C05455=1067.841,-44.416,-61.846,172.334,24.240,154.436
C05456=1067.835,-44.665,-61.833,172.333,24.238,154.436
C05457=1067.828,-44.914,-61.820,172.331,24.236,154.436
C05458=1067.822,-45.164,-61.808,172.330,24.234,154.436
C05459=1067.816,-45.414,-61.795,172.328,24.232,154.436
C05460=1067.810,-45.664,-61.783,172.327,24.229,154.435
C05461=1067.804,-45.913,-61.771,172.325,24.227,154.435
C05462=1067.798,-46.163,-61.759,172.324,24.225,154.435
C05463=1067.792,-46.413,-61.746,172.322,24.223,154.435
C05464=1067.786,-46.662,-61.734,172.321,24.221,154.435
C05465=1067.780,-46.912,-61.722,172.320,24.219,154.434
C05466=1067.774,-47.161,-61.709,172.318,24.217,154.434
C05467=1067.768,-47.411,-61.697,172.317,24.215,154.434
C05468=1067.762,-47.661,-61.685,172.315,24.213,154.434
C05469=1067.756,-47.911,-61.672,172.313,24.211,154.434
C05470=1067.749,-48.160,-61.660,172.311,24.208,154.433
C05471=1067.744,-48.409,-61.648,172.310,24.207,154.433
C05472=1067.738,-48.659,-61.636,172.308,24.205,154.433
C05473=1067.732,-48.909,-61.623,172.307,24.202,154.433
C05474=1067.726,-49.159,-61.611,172.305,24.200,154.433
C05475=1067.720,-49.408,-61.599,172.304,24.198,154.432
C05476=1067.713,-49.686,-61.585,172.303,24.196,154.432
C05477=1067.707,-49.963,-61.572,172.301,24.194,154.432
C05478=1067.700,-50.241,-61.558,172.299,24.192,154.432
C05479=1067.693,-50.518,-61.544,172.297,24.189,154.432
C05480=1067.687,-50.767,-61.532,172.296,24.187,154.431
C05481=1067.681,-51.017,-61.520,172.294,24.186,154.431
C05482=1067.674,-51.267,-61.508,172.293,24.184,154.431
C05483=1067.668,-51.516,-61.497,172.292,24.181,154.431
C05484=1067.662,-51.766,-61.484,172.290,24.179,154.431
C05485=1067.656,-52.016,-61.472,172.289,24.178,154.431
C05486=1067.650,-52.266,-61.460,172.287,24.176,154.430
C05487=1067.643,-52.515,-61.448,172.285,24.174,154.430
C05488=1067.637,-52.764,-61.436,172.283,24.172,154.430
C05489=1067.631,-53.014,-61.424,172.282,24.169,154.430
C05490=1067.625,-53.263,-61.412,172.280,24.168,154.430
C05491=1067.618,-53.514,-61.401,172.279,24.166,154.430
C05492=1067.612,-53.764,-61.388,172.277,24.164,154.430
C05493=1067.606,-54.012,-61.376,172.276,24.162,154.429
C05494=1067.600,-54.262,-61.364,172.274,24.160,154.429
C05495=1067.594,-54.512,-61.352,172.273,24.158,154.429
C05496=1067.587,-54.762,-61.341,172.271,24.157,154.429
C05497=1067.582,-55.011,-61.328,172.270,24.154,154.429
C05498=1067.576,-55.261,-61.316,172.268,24.152,154.429
C05499=1067.569,-55.510,-61.305,172.267,24.150,154.428
C05500=1067.563,-55.760,-61.292,172.265,24.149,154.428
C05501=1067.557,-56.010,-61.281,172.264,24.147,154.428
C05502=1067.551,-56.259,-61.269,172.262,24.145,154.428
C05503=1067.545,-56.509,-61.257,172.261,24.143,154.428
C05504=1067.538,-56.759,-61.245,172.259,24.141,154.428
C05505=1067.532,-57.008,-61.234,172.258,24.139,154.427
C05506=1067.526,-57.258,-61.221,172.255,24.137,154.427
C05507=1067.520,-57.508,-61.209,172.254,24.135,154.427
C05508=1067.514,-57.757,-61.198,172.252,24.133,154.427
C05509=1067.508,-58.007,-61.186,172.251,24.131,154.427
C05510=1067.501,-58.257,-61.174,172.249,24.129,154.427
C05511=1067.495,-58.505,-61.162,172.248,24.127,154.427
C05512=1067.490,-58.756,-61.150,172.246,24.126,154.426
C05513=1067.483,-59.006,-61.138,172.245,24.124,154.426
C05514=1067.477,-59.254,-61.127,172.243,24.122,154.426
C05515=1067.471,-59.505,-61.115,172.242,24.120,154.426
C05516=1067.465,-59.755,-61.103,172.240,24.118,154.426
C05517=1067.459,-60.003,-61.091,172.239,24.116,154.426
C05518=1067.453,-60.254,-61.080,172.237,24.115,154.426
C05519=1067.447,-60.503,-61.068,172.236,24.113,154.425
C05520=1067.441,-60.752,-61.056,172.234,24.111,154.425
C05521=1067.434,-61.003,-61.045,172.233,24.109,154.425
C05522=1067.428,-61.252,-61.032,172.231,24.107,154.425
C05523=1067.423,-61.502,-61.021,172.230,24.105,154.425
C05524=1067.416,-61.751,-61.009,172.227,24.103,154.425
C05525=1067.410,-62.001,-60.997,172.226,24.101,154.425
C05526=1067.404,-62.251,-60.986,172.224,24.099,154.424
C05527=1067.398,-62.500,-60.974,172.223,24.098,154.424
C05528=1067.392,-62.750,-60.963,172.221,24.096,154.424
C05529=1067.386,-63.000,-60.951,172.220,24.094,154.424
C05530=1067.380,-63.250,-60.939,172.218,24.092,154.424
C05531=1067.374,-63.499,-60.928,172.217,24.090,154.424
C05532=1067.368,-63.749,-60.916,172.215,24.088,154.424
C05533=1067.362,-63.998,-60.904,172.214,24.087,154.423
C05534=1067.356,-64.248,-60.893,172.212,24.085,154.423
C05535=1067.350,-64.497,-60.881,172.211,24.083,154.423
C05536=1067.344,-64.748,-60.870,172.209,24.081,154.423
C05537=1067.337,-64.997,-60.858,172.208,24.079,154.423
C05538=1067.332,-65.247,-60.847,172.206,24.077,154.423
C05539=1067.325,-65.496,-60.835,172.205,24.076,154.423
C05540=1067.319,-65.775,-60.822,172.202,24.073,154.422
C05541=1067.312,-66.054,-60.809,172.201,24.071,154.422
C05542=1067.305,-66.332,-60.797,172.199,24.069,154.422
C05543=1067.299,-66.611,-60.784,172.198,24.067,154.422
C05544=1067.292,-66.861,-60.772,172.196,24.065,154.422
C05545=1067.287,-67.111,-60.760,172.194,24.063,154.422
C05546=1067.280,-67.360,-60.748,172.192,24.062,154.422
C05547=1067.275,-67.610,-60.738,172.191,24.060,154.422
C05548=1067.268,-67.859,-60.726,172.189,24.058,154.421
C05549=1067.262,-68.109,-60.715,172.188,24.056,154.421
C05550=1067.257,-68.359,-60.703,172.186,24.055,154.421
C05551=1067.251,-68.608,-60.691,172.185,24.053,154.421
C05552=1067.244,-68.858,-60.680,172.183,24.051,154.421
C05553=1067.238,-69.107,-60.668,172.182,24.049,154.421
C05554=1067.232,-69.357,-60.657,172.180,24.047,154.421
C05555=1067.227,-69.607,-60.646,172.179,24.045,154.420
C05556=1067.220,-69.857,-60.634,172.177,24.044,154.420
C05557=1067.214,-70.106,-60.623,172.175,24.042,154.420
C05558=1067.208,-70.357,-60.612,172.174,24.040,154.420
C05559=1067.202,-70.605,-60.600,172.172,24.038,154.420
C05560=1067.196,-70.856,-60.588,172.171,24.037,154.420
C05561=1067.191,-71.105,-60.577,172.169,24.035,154.420
C05562=1067.184,-71.355,-60.565,172.168,24.033,154.419
C05563=1067.178,-71.604,-60.554,172.166,24.032,154.419
C05564=1067.173,-71.854,-60.544,172.165,24.030,154.419
C05565=1067.167,-72.104,-60.531,172.163,24.028,154.419
C05566=1067.161,-72.353,-60.520,172.161,24.026,154.419
C05567=1067.155,-72.604,-60.509,172.159,24.024,154.419
C05568=1067.149,-72.853,-60.498,172.158,24.022,154.419
C05569=1067.142,-73.103,-60.486,172.156,24.021,154.419
C05570=1067.136,-73.352,-60.475,172.155,24.019,154.419
C05571=1067.131,-73.602,-60.464,172.153,24.017,154.419
C05572=1067.125,-73.852,-60.453,172.152,24.015,154.418
C05573=1067.119,-74.101,-60.441,172.150,24.013,154.418
C05574=1067.113,-74.351,-60.430,172.148,24.012,154.418
C05575=1067.107,-74.601,-60.419,172.147,24.010,154.418
C05576=1067.101,-74.851,-60.408,172.145,24.008,154.418
C05577=1067.095,-75.100,-60.397,172.144,24.007,154.418
C05578=1067.088,-75.350,-60.385,172.142,24.005,154.418
C05579=1067.082,-75.599,-60.374,172.141,24.003,154.418
C05580=1067.076,-75.849,-60.364,172.139,24.002,154.418
C05581=1067.070,-76.099,-60.352,172.138,24.000,154.417
C05582=1067.064,-76.348,-60.341,172.136,23.999,154.417
C05583=1067.058,-76.598,-60.330,172.134,23.997,154.417
C05584=1067.052,-76.847,-60.319,172.133,23.995,154.417
C05585=1067.045,-77.097,-60.307,172.131,23.994,154.417
C05586=1067.040,-77.347,-60.296,172.130,23.992,154.417
C05587=1067.034,-77.596,-60.286,172.128,23.990,154.417
C05588=1067.027,-77.847,-60.274,172.126,23.989,154.417
C05589=1067.022,-78.096,-60.263,172.124,23.987,154.417
C05590=1067.015,-78.346,-60.252,172.122,23.986,154.417
C05591=1067.010,-78.596,-60.241,172.121,23.984,154.417
C05592=1067.003,-78.845,-60.231,172.119,23.982,154.416
C05593=1066.997,-79.095,-60.220,172.118,23.981,154.416
C05594=1066.991,-79.344,-60.208,172.116,23.979,154.416
C05595=1066.985,-79.594,-60.197,172.115,23.978,154.416
C05596=1066.979,-79.844,-60.186,172.113,23.976,154.416
C05597=1066.973,-80.093,-60.175,172.111,23.974,154.416
C05598=1066.967,-80.343,-60.164,172.110,23.973,154.416
C05599=1066.960,-80.593,-60.154,172.108,23.971,154.416
C05600=1066.954,-80.843,-60.142,172.107,23.969,154.416
C05601=1066.948,-81.092,-60.132,172.105,23.968,154.416
C05602=1066.942,-81.341,-60.121,172.104,23.966,154.416
C05603=1066.935,-81.592,-60.110,172.102,23.965,154.416
C05604=1066.929,-81.873,-60.098,172.100,23.963,154.415
C05605=1066.922,-82.154,-60.086,172.098,23.962,154.416
C05606=1066.915,-82.435,-60.073,172.096,23.960,154.415
C05607=1066.908,-82.715,-60.062,172.095,23.958,154.415
C05608=1066.902,-82.965,-60.051,172.093,23.957,154.415
C05609=1066.895,-83.215,-60.040,172.092,23.955,154.415
C05610=1066.889,-83.464,-60.029,172.090,23.953,154.415
C05611=1066.883,-83.714,-60.018,172.088,23.952,154.415
C05612=1066.877,-83.964,-60.007,172.086,23.951,154.415
C05613=1066.870,-84.213,-59.997,172.084,23.949,154.415
C05614=1066.864,-84.463,-59.986,172.083,23.947,154.415
C05615=1066.858,-84.713,-59.975,172.081,23.946,154.415
C05616=1066.853,-84.963,-59.965,172.079,23.944,154.415
C05617=1066.846,-85.213,-59.954,172.078,23.943,154.415
C05618=1066.840,-85.462,-59.943,172.076,23.942,154.415
C05619=1066.834,-85.712,-59.932,172.075,23.940,154.415
C05620=1066.827,-85.961,-59.922,172.073,23.939,154.415
C05621=1066.822,-86.211,-59.911,172.071,23.937,154.414
C05622=1066.816,-86.460,-59.900,172.070,23.935,154.414
C05623=1066.809,-86.710,-59.889,172.068,23.934,154.414
C05624=1066.803,-86.960,-59.879,172.066,23.933,154.414
C05625=1066.797,-87.210,-59.869,172.065,23.931,154.414
C05626=1066.791,-87.459,-59.858,172.063,23.930,154.414
C05627=1066.785,-87.709,-59.847,172.062,23.928,154.414
C05628=1066.778,-87.958,-59.836,172.060,23.927,154.414
C05629=1066.773,-88.208,-59.826,172.058,23.925,154.414
C05630=1066.766,-88.459,-59.815,172.057,23.924,154.414
C05631=1066.760,-88.708,-59.805,172.055,23.922,154.414
C05632=1066.754,-88.957,-59.794,172.054,23.921,154.414
C05633=1066.749,-89.207,-59.783,172.052,23.920,154.414
C05634=1066.742,-89.457,-59.773,172.050,23.918,154.414
C05635=1066.736,-89.707,-59.762,172.049,23.916,154.414
C05636=1066.730,-89.956,-59.752,172.047,23.915,154.414
C05637=1066.724,-90.206,-59.741,172.046,23.914,154.414
C05638=1066.718,-90.456,-59.730,172.044,23.913,154.414
C05639=1066.711,-90.706,-59.720,172.042,23.911,154.414
C05640=1066.706,-90.955,-59.709,172.041,23.909,154.413
C05641=1066.700,-91.205,-59.698,172.039,23.908,154.413
C05642=1066.693,-91.455,-59.689,172.037,23.907,154.413
C05643=1066.687,-91.705,-59.678,172.036,23.905,154.413
C05644=1066.681,-91.954,-59.667,172.033,23.903,154.413
C05645=1066.675,-92.204,-59.657,172.032,23.902,154.413
C05646=1066.670,-92.453,-59.646,172.030,23.901,154.413
C05647=1066.663,-92.703,-59.636,172.028,23.900,154.413
C05648=1066.657,-92.953,-59.626,172.027,23.898,154.413
C05649=1066.651,-93.203,-59.615,172.025,23.896,154.413
C05650=1066.645,-93.452,-59.604,172.023,23.895,154.413
C05651=1066.639,-93.702,-59.595,172.022,23.894,154.413
C05652=1066.633,-93.951,-59.584,172.020,23.893,154.413
C05653=1066.627,-94.201,-59.573,172.018,23.891,154.413
C05654=1066.620,-94.451,-59.563,172.017,23.889,154.413
C05655=1066.615,-94.701,-59.552,172.015,23.888,154.413
C05656=1066.608,-94.950,-59.542,172.014,23.887,154.413
C05657=1066.603,-95.200,-59.532,172.012,23.886,154.413
C05658=1066.596,-95.449,-59.521,172.010,23.884,154.413
C05659=1066.590,-95.700,-59.511,172.009,23.883,154.413
C05660=1066.585,-95.950,-59.500,172.007,23.881,154.413
C05661=1066.578,-96.199,-59.490,172.006,23.880,154.413
C05662=1066.573,-96.449,-59.480,172.004,23.879,154.413
C05663=1066.566,-96.698,-59.469,172.002,23.877,154.413
C05664=1066.561,-96.948,-59.459,172.001,23.876,154.413
C05665=1066.554,-97.197,-59.449,171.999,23.875,154.413
C05666=1066.549,-97.447,-59.439,171.997,23.873,154.413
C05667=1066.542,-97.697,-59.428,171.996,23.872,154.413
C05668=1066.535,-97.980,-59.416,171.994,23.871,154.413
C05669=1066.528,-98.264,-59.405,171.991,23.869,154.413
C05670=1066.521,-98.547,-59.393,171.990,23.868,154.413
C05671=1066.514,-98.830,-59.381,171.988,23.866,154.412
C05672=1066.508,-99.080,-59.372,171.986,23.865,154.413
C05673=1066.501,-99.329,-59.362,171.985,23.864,154.413
C05674=1066.496,-99.579,-59.351,171.983,23.863,154.413
C05675=1066.490,-99.828,-59.341,171.981,23.862,154.413
C05676=1066.484,-100.079,-59.331,171.980,23.860,154.413
C05677=1066.477,-100.329,-59.321,171.978,23.859,154.413
C05678=1066.471,-100.578,-59.311,171.976,23.858,154.413
C05679=1066.465,-100.828,-59.301,171.975,23.856,154.412
C05680=1066.459,-101.078,-59.290,171.973,23.855,154.412
C05681=1066.453,-101.327,-59.281,171.971,23.854,154.412
C05682=1066.446,-101.576,-59.271,171.970,23.853,154.412
C05683=1066.441,-101.827,-59.260,171.968,23.851,154.412
C05684=1066.435,-102.076,-59.251,171.966,23.851,154.413
C05685=1066.428,-102.326,-59.240,171.965,23.849,154.413
C05686=1066.422,-102.576,-59.230,171.963,23.848,154.413
C05687=1066.416,-102.826,-59.220,171.961,23.847,154.412
C05688=1066.410,-103.075,-59.210,171.960,23.845,154.412
C05689=1066.404,-103.325,-59.200,171.958,23.844,154.412
C05690=1066.398,-103.575,-59.190,171.956,23.843,154.412
C05691=1066.391,-103.824,-59.180,171.954,23.842,154.413
C05692=1066.386,-104.075,-59.170,171.953,23.841,154.413
C05693=1066.380,-104.324,-59.160,171.951,23.840,154.413
C05694=1066.373,-104.574,-59.150,171.949,23.838,154.413
C05695=1066.367,-104.823,-59.141,171.948,23.837,154.413
C05696=1066.361,-105.073,-59.130,171.946,23.836,154.412
C05697=1066.355,-105.323,-59.120,171.944,23.835,154.413
C05698=1066.349,-105.572,-59.111,171.943,23.834,154.413
C05699=1066.343,-105.822,-59.100,171.941,23.832,154.413
C05700=1066.337,-106.072,-59.090,171.939,23.831,154.413
C05701=1066.331,-106.321,-59.081,171.938,23.830,154.413
C05702=1066.325,-106.571,-59.071,171.936,23.829,154.413
C05703=1066.318,-106.820,-59.061,171.934,23.828,154.413
C05704=1066.312,-107.071,-59.050,171.933,23.827,154.413
C05705=1066.306,-107.321,-59.041,171.931,23.826,154.413
C05706=1066.300,-107.571,-59.031,171.929,23.825,154.413
C05707=1066.294,-107.820,-59.021,171.927,23.823,154.413
C05708=1066.287,-108.070,-59.011,171.926,23.823,154.413
C05709=1066.281,-108.320,-59.002,171.924,23.821,154.413
C05710=1066.275,-108.569,-58.992,171.922,23.820,154.413
C05711=1066.269,-108.819,-58.981,171.920,23.819,154.413
C05712=1066.263,-109.069,-58.972,171.919,23.818,154.413
C05713=1066.257,-109.319,-58.962,171.917,23.817,154.413
C05714=1066.251,-109.568,-58.952,171.915,23.816,154.413
C05715=1066.245,-109.818,-58.943,171.914,23.815,154.413
C05716=1066.238,-110.068,-58.933,171.912,23.813,154.413
C05717=1066.232,-110.317,-58.923,171.910,23.813,154.413
C05718=1066.226,-110.567,-58.913,171.909,23.811,154.413
C05719=1066.220,-110.817,-58.904,171.907,23.811,154.413
C05720=1066.214,-111.067,-58.894,171.905,23.809,154.413
C05721=1066.208,-111.317,-58.884,171.903,23.808,154.413
C05722=1066.202,-111.566,-58.875,171.902,23.807,154.413
C05723=1066.196,-111.816,-58.865,171.900,23.806,154.413
C05724=1066.189,-112.065,-58.855,171.898,23.805,154.413
C05725=1066.183,-112.315,-58.845,171.896,23.804,154.413
C05726=1066.177,-112.565,-58.836,171.895,23.803,154.413
C05727=1066.171,-112.815,-58.826,171.893,23.802,154.413
C05728=1066.165,-113.065,-58.816,171.891,23.801,154.413
C05729=1066.158,-113.314,-58.807,171.889,23.800,154.414
C05730=1066.153,-113.563,-58.798,171.888,23.799,154.414
C05731=1066.147,-113.813,-58.788,171.886,23.798,154.414
C05732=1066.140,-114.095,-58.776,171.883,23.797,154.414
C05733=1066.133,-114.376,-58.766,171.882,23.796,154.414
C05734=1066.126,-114.657,-58.755,171.880,23.795,154.414
C05735=1066.119,-114.939,-58.744,171.878,23.794,154.414
C05736=1066.113,-115.188,-58.735,171.876,23.793,154.414
C05737=1066.107,-115.438,-58.725,171.875,23.792,154.414
C05738=1066.101,-115.687,-58.716,171.873,23.791,154.414
C05739=1066.095,-115.937,-58.706,171.871,23.790,154.414
C05740=1066.088,-116.187,-58.696,171.870,23.789,154.414
C05741=1066.082,-116.437,-58.687,171.868,23.788,154.414
C05742=1066.076,-116.687,-58.677,171.866,23.787,154.414
C05743=1066.070,-116.936,-58.668,171.864,23.786,154.414
C05744=1066.064,-117.186,-58.658,171.862,23.785,154.414
C05745=1066.058,-117.436,-58.649,171.861,23.784,154.414
C05746=1066.051,-117.686,-58.639,171.859,23.783,154.414
C05747=1066.044,-117.935,-58.630,171.857,23.782,154.415
C05748=1066.039,-118.186,-58.621,171.855,23.781,154.415
C05749=1066.033,-118.435,-58.612,171.854,23.780,154.415
C05750=1066.027,-118.685,-58.602,171.852,23.780,154.415
C05751=1066.021,-118.934,-58.593,171.850,23.778,154.415
C05752=1066.015,-119.184,-58.583,171.848,23.778,154.415
C05753=1066.008,-119.434,-58.574,171.847,23.777,154.415
C05754=1066.002,-119.684,-58.564,171.845,23.776,154.415
C05755=1065.996,-119.934,-58.555,171.843,23.775,154.415
C05756=1065.990,-120.183,-58.545,171.841,23.774,154.415
C05757=1065.984,-120.432,-58.536,171.840,23.773,154.415
C05758=1065.978,-120.683,-58.528,171.838,23.772,154.415
C05759=1065.971,-120.932,-58.518,171.836,23.772,154.415
C05760=1065.965,-121.182,-58.508,171.834,23.770,154.415
C05761=1065.959,-121.432,-58.499,171.832,23.770,154.416
C05762=1065.953,-121.682,-58.489,171.831,23.769,154.416
C05763=1065.947,-121.932,-58.480,171.829,23.768,154.416
C05764=1065.941,-122.181,-58.471,171.827,23.767,154.416
C05765=1065.935,-122.431,-58.462,171.825,23.766,154.416
C05766=1065.928,-122.681,-58.453,171.823,23.765,154.416
C05767=1065.922,-122.930,-58.443,171.822,23.765,154.416
C05768=1065.916,-123.180,-58.434,171.820,23.764,154.416
C05769=1065.910,-123.430,-58.424,171.818,23.763,154.416
C05770=1065.905,-123.680,-58.416,171.816,23.762,154.416
C05771=1065.898,-123.929,-58.407,171.815,23.762,154.416
C05772=1065.892,-124.179,-58.397,171.814,23.761,154.416
C05773=1065.885,-124.429,-58.387,171.812,23.760,154.416
C05774=1065.880,-124.679,-58.379,171.810,23.759,154.417
C05775=1065.873,-124.929,-58.369,171.808,23.758,154.417
C05776=1065.867,-125.178,-58.360,171.807,23.757,154.417
C05777=1065.861,-125.428,-58.351,171.805,23.757,154.417
C05778=1065.855,-125.678,-58.342,171.803,23.756,154.417
C05779=1065.849,-125.928,-58.332,171.801,23.755,154.417
C05780=1065.842,-126.177,-58.323,171.799,23.755,154.417
C05781=1065.837,-126.427,-58.315,171.797,23.754,154.417
C05782=1065.831,-126.677,-58.305,171.796,23.753,154.417
C05783=1065.824,-126.926,-58.296,171.794,23.752,154.417
C05784=1065.817,-127.176,-58.287,171.792,23.751,154.418
C05785=1065.812,-127.427,-58.278,171.790,23.750,154.418
C05786=1065.805,-127.675,-58.269,171.788,23.750,154.418
C05787=1065.799,-127.925,-58.260,171.787,23.749,154.418
C05788=1065.795,-128.176,-58.250,171.785,23.748,154.418
C05789=1065.792,-128.427,-58.239,171.784,23.746,154.418
C05790=1065.791,-128.678,-58.228,171.782,23.743,154.417
C05791=1065.791,-128.928,-58.215,171.781,23.740,154.417
C05792=1065.794,-129.181,-58.202,171.781,23.736,154.416
C05793=1065.798,-129.433,-58.189,171.781,23.731,154.416
C05794=1065.804,-129.683,-58.175,171.780,23.726,154.415
C05795=1065.811,-129.934,-58.159,171.780,23.720,154.414
C05796=1065.426,-129.956,-58.337,171.733,23.868,154.446
C05797=1065.418,-129.706,-58.353,171.733,23.875,154.447
C05798=1065.412,-129.455,-58.368,171.733,23.880,154.448
C05799=1065.409,-129.203,-58.381,171.733,23.884,154.449
C05800=1065.406,-128.951,-58.395,171.734,23.888,154.450
C05801=1065.406,-128.700,-58.406,171.735,23.892,154.450
C05802=1065.406,-128.450,-58.418,171.737,23.895,154.451
C05803=1065.410,-128.199,-58.429,171.738,23.896,154.451
C05804=1065.414,-127.948,-58.439,171.740,23.898,154.451
C05805=1065.419,-127.698,-58.448,171.742,23.898,154.451
C05806=1065.426,-127.448,-58.457,171.743,23.900,154.451
C05807=1065.432,-127.198,-58.467,171.745,23.900,154.450
C05808=1065.438,-126.950,-58.475,171.747,23.901,154.450
C05809=1065.444,-126.699,-58.484,171.749,23.902,154.450
C05810=1065.450,-126.449,-58.494,171.751,23.903,154.450
C05811=1065.457,-126.200,-58.503,171.751,23.903,154.450
C05812=1065.462,-125.950,-58.511,171.753,23.904,154.450
C05813=1065.468,-125.700,-58.521,171.755,23.904,154.450
C05814=1065.475,-125.451,-58.530,171.757,23.905,154.450
C05815=1065.482,-125.201,-58.539,171.759,23.906,154.450
C05816=1065.487,-124.951,-58.548,171.761,23.906,154.449
C05817=1065.494,-124.701,-58.558,171.762,23.908,154.450
C05818=1065.499,-124.452,-58.567,171.764,23.908,154.449
C05819=1065.506,-124.202,-58.576,171.766,23.909,154.449
C05820=1065.512,-123.952,-58.585,171.768,23.910,154.449
C05821=1065.518,-123.702,-58.594,171.769,23.911,154.449
C05822=1065.524,-123.452,-58.604,171.771,23.912,154.449
C05823=1065.530,-123.203,-58.613,171.773,23.913,154.449
C05824=1065.536,-122.953,-58.623,171.775,23.913,154.449
C05825=1065.543,-122.703,-58.631,171.777,23.914,154.449
C05826=1065.549,-122.454,-58.640,171.778,23.915,154.449
C05827=1065.555,-122.204,-58.650,171.780,23.916,154.449
C05828=1065.561,-121.954,-58.660,171.782,23.917,154.449
C05829=1065.567,-121.704,-58.669,171.784,23.917,154.448
C05830=1065.573,-121.454,-58.678,171.786,23.918,154.448
C05831=1065.579,-121.205,-58.687,171.787,23.919,154.448
C05832=1065.586,-120.955,-58.696,171.789,23.920,154.448
C05833=1065.592,-120.705,-58.706,171.791,23.921,154.448
C05834=1065.598,-120.456,-58.715,171.793,23.922,154.448
C05835=1065.604,-120.206,-58.725,171.794,23.923,154.448
C05836=1065.610,-119.956,-58.734,171.796,23.923,154.448
C05837=1065.616,-119.707,-58.744,171.798,23.924,154.448
C05838=1065.622,-119.456,-58.753,171.800,23.925,154.448
C05839=1065.628,-119.207,-58.762,171.802,23.926,154.448
C05840=1065.634,-118.957,-58.772,171.803,23.927,154.448
C05841=1065.641,-118.707,-58.781,171.805,23.928,154.448
C05842=1065.647,-118.458,-58.790,171.807,23.929,154.447
C05843=1065.653,-118.208,-58.800,171.808,23.930,154.447
C05844=1065.660,-117.958,-58.809,171.810,23.931,154.447
C05845=1065.666,-117.708,-58.819,171.812,23.931,154.447
C05846=1065.672,-117.458,-58.828,171.814,23.933,154.447
C05847=1065.677,-117.209,-58.838,171.816,23.933,154.447
C05848=1065.684,-116.959,-58.847,171.817,23.934,154.447
C05849=1065.690,-116.710,-58.857,171.819,23.935,154.447
C05850=1065.696,-116.460,-58.866,171.821,23.936,154.447
C05851=1065.702,-116.210,-58.876,171.823,23.937,154.447
C05852=1065.708,-115.960,-58.885,171.824,23.938,154.447
C05853=1065.714,-115.740,-58.893,171.825,23.938,154.447
C05854=1065.719,-115.520,-58.902,171.827,23.940,154.447
C05855=1065.725,-115.300,-58.910,171.829,23.940,154.447
C05856=1065.730,-115.080,-58.919,171.830,23.942,154.447
C05857=1065.736,-114.860,-58.927,171.831,23.942,154.447
C05858=1065.741,-114.639,-58.936,171.833,23.943,154.447
C05859=1065.747,-114.420,-58.944,171.835,23.944,154.447
C05860=1065.751,-114.199,-58.952,171.837,23.945,154.446
C05861=1065.761,-113.836,-58.966,171.839,23.946,154.446
C05862=1065.767,-113.586,-58.976,171.841,23.948,154.446
C05863=1065.773,-113.336,-58.985,171.843,23.948,154.446
C05864=1065.779,-113.086,-58.996,171.844,23.950,154.446
C05865=1065.785,-112.836,-59.005,171.846,23.950,154.446
C05866=1065.791,-112.587,-59.015,171.848,23.952,154.446
C05867=1065.797,-112.337,-59.024,171.850,23.952,154.446
C05868=1065.804,-112.088,-59.035,171.851,23.954,154.446
C05869=1065.810,-111.838,-59.044,171.853,23.955,154.446
C05870=1065.816,-111.588,-59.054,171.855,23.956,154.446
C05871=1065.822,-111.338,-59.063,171.857,23.957,154.446
C05872=1065.828,-111.089,-59.073,171.858,23.958,154.446
C05873=1065.834,-110.839,-59.082,171.860,23.959,154.446
C05874=1065.841,-110.589,-59.092,171.862,23.960,154.446
C05875=1065.846,-110.339,-59.103,171.864,23.961,154.446
C05876=1065.852,-110.090,-59.112,171.865,23.962,154.446
C05877=1065.859,-109.840,-59.122,171.867,23.963,154.446
C05878=1065.865,-109.590,-59.132,171.869,23.964,154.446
C05879=1065.871,-109.340,-59.141,171.870,23.965,154.446
C05880=1065.877,-109.090,-59.151,171.872,23.966,154.446
C05881=1065.884,-108.841,-59.161,171.874,23.967,154.446
C05882=1065.890,-108.591,-59.171,171.876,23.969,154.446
C05883=1065.896,-108.342,-59.180,171.877,23.969,154.446
C05884=1065.901,-108.092,-59.190,171.879,23.971,154.446
C05885=1065.908,-107.842,-59.201,171.881,23.972,154.446
C05886=1065.914,-107.593,-59.210,171.883,23.973,154.446
C05887=1065.920,-107.343,-59.220,171.884,23.974,154.446
C05888=1065.926,-107.093,-59.229,171.886,23.975,154.446
C05889=1065.933,-106.843,-59.239,171.888,23.976,154.445
C05890=1065.938,-106.594,-59.250,171.889,23.977,154.445
C05891=1065.944,-106.344,-59.259,171.891,23.978,154.445
C05892=1065.951,-106.094,-59.269,171.893,23.980,154.445
C05893=1065.957,-105.845,-59.279,171.894,23.980,154.445
C05894=1065.963,-105.595,-59.289,171.896,23.982,154.445
C05895=1065.969,-105.345,-59.299,171.898,23.983,154.445
C05896=1065.976,-105.095,-59.309,171.899,23.984,154.445
C05897=1065.982,-104.845,-59.319,171.901,23.986,154.445
C05898=1065.987,-104.595,-59.329,171.903,23.986,154.445
C05899=1065.994,-104.345,-59.339,171.905,23.988,154.445
C05900=1066.000,-104.096,-59.349,171.906,23.989,154.445
C05901=1066.006,-103.846,-59.359,171.908,23.990,154.445
C05902=1066.012,-103.597,-59.370,171.910,23.991,154.445
C05903=1066.018,-103.347,-59.379,171.911,23.993,154.445
C05904=1066.024,-103.097,-59.389,171.913,23.993,154.445
C05905=1066.030,-102.848,-59.400,171.915,23.995,154.445
C05906=1066.036,-102.598,-59.409,171.916,23.996,154.445
C05907=1066.042,-102.348,-59.419,171.918,23.997,154.445
C05908=1066.048,-102.099,-59.430,171.920,23.998,154.445
C05909=1066.055,-101.848,-59.439,171.921,24.000,154.445
C05910=1066.061,-101.599,-59.450,171.923,24.001,154.445
C05911=1066.067,-101.349,-59.460,171.925,24.002,154.445
C05912=1066.073,-101.099,-59.469,171.927,24.003,154.445
C05913=1066.079,-100.850,-59.480,171.928,24.004,154.445
C05914=1066.085,-100.600,-59.490,171.930,24.006,154.445
C05915=1066.091,-100.351,-59.500,171.932,24.007,154.445
C05916=1066.098,-100.101,-59.510,171.933,24.008,154.445
C05917=1066.103,-99.851,-59.521,171.935,24.009,154.445
C05918=1066.110,-99.601,-59.531,171.937,24.011,154.445
C05919=1066.117,-99.352,-59.541,171.938,24.012,154.445
C05920=1066.122,-99.102,-59.551,171.940,24.013,154.445
C05921=1066.128,-98.853,-59.561,171.942,24.015,154.445
C05922=1066.135,-98.569,-59.572,171.943,24.016,154.445
C05923=1066.143,-98.286,-59.584,171.946,24.017,154.445
C05924=1066.149,-98.003,-59.596,171.948,24.019,154.445
C05925=1066.156,-97.719,-59.607,171.949,24.020,154.445
C05926=1066.163,-97.469,-59.618,171.951,24.021,154.445
C05927=1066.168,-97.219,-59.628,171.953,24.023,154.445
C05928=1066.175,-96.970,-59.638,171.954,24.024,154.445
C05929=1066.180,-96.720,-59.648,171.956,24.026,154.446
C05930=1066.187,-96.471,-59.659,171.957,24.027,154.446
C05931=1066.192,-96.221,-59.670,171.959,24.028,154.446
C05932=1066.199,-95.971,-59.679,171.961,24.029,154.446
C05933=1066.204,-95.722,-59.690,171.962,24.031,154.446
C05934=1066.210,-95.471,-59.701,171.964,24.032,154.446
C05935=1066.217,-95.222,-59.711,171.966,24.033,154.446
C05936=1066.223,-94.972,-59.722,171.967,24.035,154.446
C05937=1066.229,-94.722,-59.731,171.969,24.036,154.446
C05938=1066.235,-94.473,-59.742,171.971,24.038,154.446
C05939=1066.241,-94.223,-59.752,171.972,24.039,154.446
C05940=1066.247,-93.973,-59.763,171.974,24.040,154.446
C05941=1066.253,-93.724,-59.774,171.976,24.042,154.446
C05942=1066.259,-93.474,-59.783,171.978,24.043,154.446
C05943=1066.265,-93.224,-59.794,171.980,24.045,154.446
C05944=1066.271,-92.975,-59.805,171.981,24.046,154.446
C05945=1066.277,-92.724,-59.815,171.983,24.048,154.446
C05946=1066.284,-92.475,-59.825,171.985,24.049,154.446
C05947=1066.289,-92.226,-59.836,171.986,24.050,154.446
C05948=1066.295,-91.975,-59.846,171.988,24.052,154.446
C05949=1066.301,-91.726,-59.857,171.989,24.053,154.446
C05950=1066.308,-91.476,-59.868,171.991,24.054,154.446
C05951=1066.314,-91.226,-59.878,171.993,24.056,154.446
C05952=1066.320,-90.977,-59.888,171.994,24.058,154.446
C05953=1066.325,-90.727,-59.899,171.996,24.059,154.446
C05954=1066.332,-90.478,-59.910,171.998,24.060,154.446
C05955=1066.338,-90.227,-59.920,171.999,24.061,154.446
C05956=1066.344,-89.978,-59.931,172.001,24.063,154.447
C05957=1066.350,-89.729,-59.941,172.002,24.065,154.447
C05958=1066.356,-89.479,-59.952,172.004,24.066,154.447
C05959=1066.363,-89.229,-59.962,172.006,24.067,154.447
C05960=1066.368,-88.979,-59.973,172.007,24.069,154.447
C05961=1066.374,-88.730,-59.984,172.009,24.070,154.447
C05962=1066.381,-88.480,-59.995,172.011,24.072,154.447
C05963=1066.387,-88.230,-60.005,172.012,24.073,154.447
C05964=1066.392,-87.980,-60.016,172.014,24.075,154.447
C05965=1066.399,-87.731,-60.026,172.016,24.076,154.447
C05966=1066.405,-87.481,-60.037,172.017,24.077,154.447
C05967=1066.411,-87.231,-60.048,172.019,24.079,154.447
C05968=1066.417,-86.982,-60.058,172.020,24.080,154.447
C05969=1066.424,-86.732,-60.069,172.022,24.082,154.447
C05970=1066.430,-86.482,-60.079,172.024,24.083,154.447
C05971=1066.436,-86.233,-60.090,172.025,24.085,154.447
C05972=1066.442,-85.982,-60.101,172.027,24.086,154.447
C05973=1066.448,-85.733,-60.111,172.028,24.088,154.448
C05974=1066.454,-85.484,-60.122,172.031,24.089,154.447
C05975=1066.460,-85.234,-60.134,172.033,24.091,154.448
C05976=1066.467,-84.984,-60.144,172.034,24.093,154.448
C05977=1066.473,-84.735,-60.155,172.036,24.094,154.448
C05978=1066.479,-84.485,-60.166,172.037,24.096,154.448
C05979=1066.484,-84.235,-60.176,172.039,24.097,154.448
C05980=1066.491,-83.985,-60.186,172.041,24.098,154.448
C05981=1066.497,-83.735,-60.198,172.042,24.100,154.448
C05982=1066.503,-83.486,-60.209,172.044,24.101,154.448
C05983=1066.510,-83.237,-60.219,172.046,24.103,154.448
C05984=1066.516,-82.986,-60.230,172.047,24.104,154.448
C05985=1066.522,-82.737,-60.241,172.049,24.106,154.448
C05986=1066.530,-82.456,-60.253,172.050,24.108,154.448
C05987=1066.536,-82.175,-60.265,172.053,24.109,154.448
C05988=1066.543,-81.894,-60.278,172.054,24.111,154.448
C05989=1066.550,-81.613,-60.290,172.056,24.113,154.449
C05990=1066.556,-81.363,-60.300,172.057,24.114,154.449
C05991=1066.563,-81.113,-60.311,172.059,24.115,154.449
C05992=1066.568,-80.864,-60.322,172.061,24.117,154.449
C05993=1066.574,-80.614,-60.333,172.062,24.119,154.449
C05994=1066.581,-80.364,-60.344,172.064,24.120,154.449
C05995=1066.587,-80.115,-60.354,172.066,24.122,154.449
C05996=1066.593,-79.865,-60.366,172.067,24.123,154.449
C05997=1066.599,-79.616,-60.377,172.069,24.125,154.449
C05998=1066.605,-79.366,-60.388,172.071,24.127,154.449
C05999=1066.611,-79.116,-60.399,172.073,24.128,154.449
C06000=1066.617,-78.867,-60.410,172.074,24.130,154.449
C06001=1066.624,-78.616,-60.421,172.076,24.132,154.449
C06002=1066.630,-78.367,-60.432,172.078,24.133,154.449
C06003=1066.636,-78.118,-60.443,172.079,24.135,154.450
C06004=1066.642,-77.868,-60.454,172.081,24.136,154.450
C06005=1066.648,-77.618,-60.465,172.082,24.138,154.450
C06006=1066.654,-77.368,-60.476,172.084,24.140,154.450
C06007=1066.660,-77.118,-60.487,172.085,24.141,154.450
C06008=1066.666,-76.870,-60.498,172.087,24.143,154.450
C06009=1066.672,-76.619,-60.510,172.088,24.145,154.450
C06010=1066.678,-76.370,-60.521,172.090,24.146,154.450
C06011=1066.684,-76.120,-60.532,172.092,24.148,154.450
C06012=1066.690,-75.870,-60.543,172.093,24.150,154.451
C06013=1066.696,-75.620,-60.554,172.095,24.151,154.451
C06014=1066.703,-75.371,-60.566,172.096,24.153,154.451
C06015=1066.708,-75.122,-60.576,172.098,24.154,154.451
C06016=1066.715,-74.871,-60.588,172.099,24.156,154.451
C06017=1066.720,-74.622,-60.599,172.101,24.158,154.451
C06018=1066.727,-74.372,-60.609,172.103,24.159,154.451
C06019=1066.733,-74.123,-60.621,172.104,24.161,154.451
C06020=1066.740,-73.873,-60.632,172.106,24.163,154.451
C06021=1066.745,-73.623,-60.643,172.108,24.165,154.451
C06022=1066.751,-73.373,-60.655,172.110,24.167,154.452
C06023=1066.757,-73.124,-60.666,172.111,24.168,154.452
C06024=1066.763,-72.875,-60.677,172.113,24.170,154.452
C06025=1066.769,-72.625,-60.688,172.114,24.172,154.452
C06026=1066.775,-72.375,-60.699,172.116,24.174,154.452
C06027=1066.781,-72.125,-60.712,172.117,24.176,154.452
C06028=1066.787,-71.876,-60.723,172.119,24.177,154.452
C06029=1066.793,-71.625,-60.734,172.121,24.179,154.452
C06030=1066.799,-71.377,-60.746,172.122,24.181,154.452
C06031=1066.805,-71.127,-60.756,172.124,24.182,154.453
C06032=1066.810,-70.877,-60.768,172.125,24.184,154.453
C06033=1066.816,-70.628,-60.780,172.127,24.186,154.453
C06034=1066.823,-70.378,-60.791,172.128,24.188,154.453
C06035=1066.828,-70.128,-60.802,172.130,24.190,154.453
C06036=1066.835,-69.878,-60.814,172.131,24.191,154.453
C06037=1066.841,-69.629,-60.825,172.133,24.193,154.453
C06038=1066.846,-69.378,-60.837,172.134,24.195,154.453
C06039=1066.853,-69.130,-60.848,172.136,24.197,154.454
C06040=1066.859,-68.879,-60.860,172.137,24.198,154.454
C06041=1066.865,-68.630,-60.870,172.139,24.200,154.454
C06042=1066.871,-68.380,-60.883,172.141,24.202,154.454
C06043=1066.876,-68.131,-60.894,172.143,24.204,154.454
C06044=1066.883,-67.881,-60.906,172.144,24.206,154.454
C06045=1066.889,-67.631,-60.917,172.146,24.208,154.454
C06046=1066.895,-67.382,-60.929,172.147,24.210,154.455
C06047=1066.900,-67.132,-60.940,172.149,24.211,154.455
C06048=1066.907,-66.882,-60.951,172.151,24.213,154.455
C06049=1066.913,-66.633,-60.963,172.152,24.215,154.455
C06050=1066.920,-66.353,-60.976,172.154,24.216,154.455
C06051=1066.926,-66.075,-60.989,172.155,24.219,154.455
C06052=1066.933,-65.796,-61.002,172.157,24.221,154.455
C06053=1066.940,-65.517,-61.014,172.159,24.223,154.455
C06054=1066.946,-65.268,-61.026,172.160,24.225,154.456
C06055=1066.951,-65.018,-61.038,172.162,24.227,154.456
C06056=1066.958,-64.768,-61.050,172.164,24.228,154.456
C06057=1066.964,-64.518,-61.061,172.165,24.230,154.456
C06058=1066.970,-64.269,-61.073,172.167,24.232,154.456
C06059=1066.976,-64.019,-61.084,172.168,24.234,154.456
C06060=1066.982,-63.770,-61.096,172.170,24.236,154.456
C06061=1066.988,-63.520,-61.107,172.171,24.238,154.457
C06062=1066.994,-63.271,-61.119,172.173,24.239,154.457
C06063=1067.000,-63.020,-61.131,172.175,24.242,154.457
C06064=1067.006,-62.771,-61.143,172.177,24.243,154.457
C06065=1067.013,-62.522,-61.154,172.178,24.245,154.457
C06066=1067.019,-62.272,-61.165,172.180,24.247,154.457
C06067=1067.024,-62.023,-61.178,172.181,24.249,154.457
C06068=1067.031,-61.772,-61.189,172.183,24.251,154.458
C06069=1067.037,-61.523,-61.201,172.184,24.253,154.458
C06070=1067.042,-61.274,-61.213,172.186,24.254,154.458
C06071=1067.049,-61.024,-61.224,172.187,24.256,154.458
C06072=1067.055,-60.774,-61.236,172.189,24.258,154.458
C06073=1067.061,-60.524,-61.247,172.190,24.260,154.458
C06074=1067.067,-60.275,-61.260,172.192,24.262,154.458
C06075=1067.074,-60.025,-61.272,172.193,24.264,154.459
C06076=1067.079,-59.776,-61.283,172.195,24.265,154.459
C06077=1067.085,-59.526,-61.295,172.196,24.267,154.459
C06078=1067.092,-59.276,-61.307,172.198,24.269,154.459
C06079=1067.098,-59.027,-61.318,172.199,24.271,154.459
C06080=1067.104,-58.777,-61.330,172.201,24.273,154.459
C06081=1067.110,-58.527,-61.342,172.202,24.275,154.459
C06082=1067.116,-58.278,-61.353,172.205,24.277,154.460
C06083=1067.122,-58.028,-61.366,172.206,24.279,154.460
C06084=1067.129,-57.778,-61.378,172.208,24.281,154.460
C06085=1067.135,-57.529,-61.389,172.209,24.283,154.460
C06086=1067.140,-57.279,-61.401,172.211,24.285,154.460
C06087=1067.147,-57.029,-61.413,172.212,24.287,154.460
C06088=1067.154,-56.780,-61.425,172.214,24.288,154.461
C06089=1067.159,-56.530,-61.437,172.215,24.290,154.461
C06090=1067.165,-56.280,-61.449,172.217,24.292,154.461
C06091=1067.172,-56.031,-61.461,172.218,24.294,154.461
C06092=1067.178,-55.781,-61.473,172.220,24.296,154.461
C06093=1067.184,-55.532,-61.485,172.221,24.298,154.461
C06094=1067.190,-55.282,-61.496,172.223,24.300,154.462
C06095=1067.196,-55.032,-61.508,172.224,24.302,154.462
C06096=1067.203,-54.782,-61.520,172.226,24.304,154.462
C06097=1067.209,-54.533,-61.532,172.227,24.305,154.462
C06098=1067.215,-54.284,-61.545,172.229,24.307,154.462
C06099=1067.221,-54.033,-61.556,172.230,24.309,154.462
C06100=1067.227,-53.783,-61.568,172.232,24.311,154.462
C06101=1067.233,-53.535,-61.580,172.234,24.314,154.463
C06102=1067.240,-53.285,-61.592,172.236,24.316,154.463
C06103=1067.246,-53.035,-61.605,172.237,24.317,154.463
C06104=1067.252,-52.786,-61.616,172.239,24.319,154.463
C06105=1067.259,-52.535,-61.628,172.240,24.321,154.463
C06106=1067.264,-52.286,-61.640,172.242,24.323,154.463
C06107=1067.270,-52.037,-61.652,172.243,24.325,154.464
C06108=1067.276,-51.787,-61.664,172.245,24.327,154.464
C06109=1067.283,-51.537,-61.676,172.246,24.329,154.464
C06110=1067.290,-51.288,-61.688,172.248,24.331,154.464
C06111=1067.295,-51.038,-61.701,172.249,24.333,154.464
C06112=1067.302,-50.789,-61.712,172.251,24.334,154.464
C06113=1067.308,-50.539,-61.725,172.252,24.337,154.465
C06114=1067.315,-50.261,-61.738,172.254,24.339,154.465
C06115=1067.321,-49.984,-61.752,172.256,24.341,154.465
C06116=1067.328,-49.706,-61.766,172.258,24.343,154.465
C06117=1067.334,-49.429,-61.779,172.259,24.346,154.465
C06118=1067.341,-49.179,-61.791,172.260,24.347,154.466
C06119=1067.347,-48.929,-61.803,172.262,24.350,154.466
C06120=1067.352,-48.680,-61.816,172.264,24.352,154.466
C06121=1067.359,-48.430,-61.828,172.266,24.354,154.466
C06122=1067.365,-48.181,-61.840,172.267,24.356,154.466
C06123=1067.370,-47.931,-61.853,172.269,24.358,154.466
C06124=1067.377,-47.681,-61.865,172.270,24.360,154.467
C06125=1067.382,-47.432,-61.877,172.272,24.362,154.467
C06126=1067.388,-47.182,-61.889,172.273,24.364,154.467
C06127=1067.394,-46.932,-61.902,172.274,24.367,154.467
C06128=1067.401,-46.683,-61.914,172.276,24.368,154.467
C06129=1067.407,-46.433,-61.926,172.277,24.371,154.468
C06130=1067.412,-46.183,-61.939,172.279,24.373,154.468
C06131=1067.419,-45.935,-61.951,172.280,24.375,154.468
C06132=1067.425,-45.685,-61.964,172.282,24.377,154.468
C06133=1067.431,-45.435,-61.976,172.283,24.379,154.468
C06134=1067.437,-45.185,-61.988,172.285,24.381,154.469
C06135=1067.443,-44.935,-62.001,172.286,24.383,154.469
C06136=1067.449,-44.686,-62.013,172.288,24.385,154.469
C06137=1067.455,-44.436,-62.026,172.289,24.387,154.469
C06138=1067.461,-44.187,-62.038,172.290,24.389,154.470
C06139=1067.467,-43.937,-62.050,172.293,24.392,154.470
C06140=1067.473,-43.688,-62.063,172.294,24.393,154.470
C06141=1067.479,-43.438,-62.076,172.296,24.396,154.470
C06142=1067.486,-43.188,-62.088,172.297,24.398,154.470
C06143=1067.491,-42.939,-62.100,172.299,24.400,154.470
C06144=1067.497,-42.689,-62.113,172.300,24.402,154.471
C06145=1067.503,-42.439,-62.125,172.302,24.404,154.471
C06146=1067.510,-42.190,-62.138,172.303,24.406,154.471
C06147=1067.516,-41.940,-62.151,172.305,24.409,154.471
C06148=1067.522,-41.690,-62.163,172.306,24.410,154.471
C06149=1067.528,-41.440,-62.176,172.307,24.413,154.472
C06150=1067.534,-41.191,-62.188,172.309,24.415,154.472
C06151=1067.541,-40.942,-62.201,172.310,24.417,154.472
C06152=1067.546,-40.692,-62.213,172.312,24.419,154.472
C06153=1067.552,-40.443,-62.226,172.313,24.421,154.472
C06154=1067.558,-40.193,-62.238,172.315,24.423,154.473
C06155=1067.565,-39.944,-62.251,172.316,24.425,154.473
C06156=1067.571,-39.694,-62.263,172.318,24.427,154.473
C06157=1067.576,-39.444,-62.276,172.319,24.429,154.473
C06158=1067.582,-39.194,-62.288,172.322,24.432,154.473
C06159=1067.589,-38.945,-62.301,172.323,24.434,154.474
C06160=1067.595,-38.695,-62.314,172.324,24.436,154.474
C06161=1067.601,-38.445,-62.326,172.326,24.438,154.474
C06162=1067.607,-38.196,-62.340,172.327,24.440,154.474
C06163=1067.613,-37.946,-62.352,172.329,24.443,154.475
C06164=1067.619,-37.696,-62.365,172.330,24.444,154.475
C06165=1067.625,-37.447,-62.378,172.332,24.447,154.475
C06166=1067.631,-37.198,-62.390,172.333,24.449,154.475
C06167=1067.637,-36.948,-62.403,172.335,24.451,154.475
C06168=1067.643,-36.699,-62.416,172.336,24.453,154.476
C06169=1067.649,-36.449,-62.428,172.337,24.456,154.476
C06170=1067.655,-36.199,-62.441,172.339,24.458,154.476
C06171=1067.661,-35.950,-62.454,172.340,24.460,154.476
C06172=1067.667,-35.700,-62.467,172.342,24.462,154.476
C06173=1067.673,-35.450,-62.479,172.343,24.464,154.477
C06174=1067.679,-35.201,-62.493,172.344,24.467,154.477
C06175=1067.685,-34.951,-62.505,172.346,24.468,154.477
C06176=1067.691,-34.702,-62.518,172.347,24.471,154.477
C06177=1067.697,-34.452,-62.531,172.349,24.473,154.478
C06178=1067.703,-34.175,-62.545,172.351,24.476,154.478
C06179=1067.710,-33.898,-62.560,172.352,24.478,154.478
C06180=1067.717,-33.621,-62.574,172.354,24.481,154.478
C06181=1067.724,-33.343,-62.588,172.356,24.483,154.479
C06182=1067.730,-33.094,-62.601,172.358,24.485,154.479
C06183=1067.736,-32.844,-62.614,172.359,24.488,154.479
C06184=1067.742,-32.594,-62.627,172.360,24.490,154.479
C06185=1067.748,-32.345,-62.640,172.362,24.492,154.480
C06186=1067.754,-32.095,-62.653,172.363,24.494,154.480
C06187=1067.760,-31.846,-62.666,172.365,24.497,154.480
C06188=1067.766,-31.596,-62.678,172.366,24.498,154.480
C06189=1067.772,-31.347,-62.692,172.368,24.501,154.481
C06190=1067.778,-31.097,-62.704,172.369,24.503,154.481
C06191=1067.785,-30.848,-62.718,172.371,24.505,154.481
C06192=1067.791,-30.598,-62.730,172.372,24.507,154.481
C06193=1067.797,-30.349,-62.743,172.373,24.510,154.481
C06194=1067.803,-30.099,-62.756,172.375,24.512,154.482
C06195=1067.809,-29.849,-62.769,172.376,24.514,154.482
C06196=1067.815,-29.600,-62.782,172.378,24.516,154.482
C06197=1067.821,-29.350,-62.795,172.379,24.519,154.482
C06198=1067.826,-29.101,-62.809,172.381,24.521,154.483
C06199=1067.832,-28.851,-62.821,172.382,24.523,154.483
C06200=1067.839,-28.601,-62.835,172.384,24.526,154.483
C06201=1067.845,-28.351,-62.848,172.386,24.528,154.483
C06202=1067.851,-28.102,-62.861,172.387,24.530,154.483
C06203=1067.858,-27.852,-62.874,172.389,24.532,154.484
C06204=1067.863,-27.603,-62.887,172.390,24.535,154.484
C06205=1067.870,-27.353,-62.900,172.391,24.537,154.484
C06206=1067.876,-27.104,-62.913,172.393,24.539,154.484
C06207=1067.882,-26.854,-62.926,172.394,24.541,154.485
C06208=1067.888,-26.605,-62.939,172.396,24.544,154.485
C06209=1067.893,-26.355,-62.953,172.397,24.546,154.485
C06210=1067.899,-26.105,-62.965,172.399,24.548,154.485
C06211=1067.906,-25.856,-62.979,172.400,24.550,154.486
C06212=1067.912,-25.606,-62.992,172.401,24.553,154.486
C06213=1067.918,-25.356,-63.006,172.403,24.555,154.486
C06214=1067.924,-25.107,-63.019,172.404,24.557,154.487
C06215=1067.930,-24.858,-63.032,172.405,24.560,154.487
C06216=1067.935,-24.607,-63.045,172.407,24.562,154.487
C06217=1067.941,-24.358,-63.058,172.408,24.564,154.487
C06218=1067.948,-24.109,-63.072,172.410,24.566,154.487
C06219=1067.954,-23.860,-63.085,172.411,24.569,154.488
C06220=1067.959,-23.609,-63.098,172.413,24.571,154.488
C06221=1067.965,-23.360,-63.111,172.415,24.574,154.488
C06222=1067.971,-23.111,-63.125,172.416,24.576,154.489
C06223=1067.977,-22.861,-63.139,172.418,24.579,154.489
C06224=1067.984,-22.611,-63.152,172.419,24.581,154.489
C06225=1067.990,-22.361,-63.165,172.420,24.583,154.489
C06226=1067.996,-22.112,-63.178,172.422,24.585,154.489
C06227=1068.001,-21.863,-63.192,172.423,24.588,154.490
C06228=1068.007,-21.613,-63.205,172.425,24.590,154.490
C06229=1068.014,-21.364,-63.218,172.426,24.592,154.490
C06230=1068.019,-21.113,-63.232,172.428,24.595,154.491
C06231=1068.026,-20.864,-63.245,172.429,24.597,154.491
C06232=1068.032,-20.615,-63.258,172.430,24.600,154.491
C06233=1068.037,-20.365,-63.272,172.432,24.602,154.491
C06234=1068.044,-20.116,-63.286,172.433,24.604,154.492
C06235=1068.050,-19.866,-63.299,172.435,24.606,154.492
C06236=1068.056,-19.616,-63.313,172.436,24.608,154.492
C06237=1068.062,-19.366,-63.326,172.437,24.611,154.492
C06238=1068.068,-19.117,-63.339,172.439,24.613,154.493
C06239=1068.073,-18.867,-63.353,172.440,24.616,154.493
C06240=1068.080,-18.618,-63.366,172.442,24.618,154.493
C06241=1068.086,-18.369,-63.379,172.443,24.620,154.493
C06242=1068.093,-18.091,-63.395,172.445,24.623,154.494
C06243=1068.099,-17.813,-63.410,172.447,24.625,154.494
C06244=1068.106,-17.534,-63.425,172.448,24.628,154.494
C06245=1068.113,-17.257,-63.440,172.449,24.631,154.495
C06246=1068.119,-17.007,-63.454,172.452,24.633,154.495
C06247=1068.125,-16.758,-63.467,172.453,24.636,154.495
C06248=1068.132,-16.508,-63.481,172.454,24.638,154.495
C06249=1068.137,-16.259,-63.495,172.456,24.641,154.496
C06250=1068.143,-16.009,-63.508,172.457,24.643,154.496
C06251=1068.150,-15.760,-63.521,172.459,24.645,154.496
C06252=1068.156,-15.510,-63.535,172.460,24.647,154.496
C06253=1068.162,-15.261,-63.549,172.461,24.650,154.497
C06254=1068.167,-15.011,-63.562,172.463,24.652,154.497
C06255=1068.174,-14.762,-63.576,172.464,24.654,154.497
C06256=1068.180,-14.511,-63.590,172.466,24.657,154.497
C06257=1068.186,-14.262,-63.603,172.467,24.659,154.498
C06258=1068.191,-14.013,-63.617,172.468,24.662,154.498
C06259=1068.198,-13.763,-63.630,172.470,24.664,154.498
C06260=1068.204,-13.513,-63.645,172.471,24.667,154.499
C06261=1068.209,-13.263,-63.658,172.472,24.669,154.499
C06262=1068.215,-13.014,-63.672,172.474,24.672,154.499
C06263=1068.221,-12.765,-63.686,172.475,24.674,154.499
C06264=1068.227,-12.515,-63.699,172.477,24.676,154.500
C06265=1068.233,-12.266,-63.714,172.478,24.679,154.500
C06266=1068.240,-12.016,-63.727,172.479,24.681,154.500
C06267=1068.245,-11.767,-63.741,172.481,24.683,154.501
C06268=1068.251,-11.517,-63.755,172.482,24.686,154.501
C06269=1068.257,-11.267,-63.768,172.484,24.688,154.501
C06270=1068.263,-11.018,-63.782,172.485,24.691,154.501
C06271=1068.269,-10.768,-63.796,172.487,24.693,154.502
C06272=1068.275,-10.519,-63.811,172.489,24.696,154.502
C06273=1068.281,-10.269,-63.824,172.490,24.699,154.502
C06274=1068.287,-10.020,-63.838,172.491,24.701,154.503
C06275=1068.293,-9.770,-63.852,172.493,24.703,154.503
C06276=1068.299,-9.520,-63.865,172.494,24.706,154.503
C06277=1068.305,-9.271,-63.879,172.496,24.708,154.503
C06278=1068.311,-9.022,-63.894,172.497,24.710,154.504
C06279=1068.317,-8.772,-63.907,172.498,24.713,154.504
C06280=1068.323,-8.522,-63.921,172.500,24.715,154.504
C06281=1068.328,-8.273,-63.935,172.501,24.718,154.504
C06282=1068.336,-8.023,-63.949,172.503,24.720,154.505
C06283=1068.341,-7.774,-63.963,172.504,24.722,154.505
C06284=1068.347,-7.525,-63.976,172.505,24.725,154.505
C06285=1068.353,-7.274,-63.991,172.507,24.728,154.506
C06286=1068.359,-7.025,-64.005,172.508,24.730,154.506
C06287=1068.365,-6.776,-64.019,172.509,24.732,154.506
C06288=1068.371,-6.526,-64.033,172.511,24.735,154.507
C06289=1068.377,-6.276,-64.047,172.512,24.737,154.507
C06290=1068.383,-6.028,-64.061,172.514,24.739,154.507
C06291=1068.389,-5.777,-64.075,172.515,24.742,154.507
C06292=1068.395,-5.528,-64.089,172.516,24.744,154.508
C06293=1068.402,-5.278,-64.103,172.518,24.747,154.508
C06294=1068.408,-5.029,-64.117,172.519,24.749,154.508
C06295=1068.413,-4.779,-64.131,172.521,24.751,154.508
C06296=1068.420,-4.530,-64.145,172.522,24.754,154.509
C06297=1068.426,-4.280,-64.159,172.523,24.757,154.509
C06298=1068.432,-4.030,-64.173,172.526,24.759,154.509
C06299=1068.438,-3.781,-64.187,172.527,24.762,154.510
C06300=1068.444,-3.532,-64.201,172.528,24.764,154.510
C06301=1068.450,-3.282,-64.216,172.530,24.766,154.510
C06302=1068.456,-3.033,-64.230,172.531,24.769,154.510
C06303=1068.462,-2.783,-64.243,172.532,24.772,154.511
C06304=1068.468,-2.534,-64.258,172.534,24.774,154.511
C06305=1068.474,-2.284,-64.272,172.535,24.776,154.511
C06306=1068.480,-2.004,-64.288,172.537,24.779,154.512
C06307=1068.487,-1.725,-64.304,172.538,24.782,154.512
C06308=1068.493,-1.446,-64.320,172.540,24.785,154.512
C06309=1068.500,-1.166,-64.336,172.541,24.788,154.513
C06310=1068.506,-0.916,-64.351,172.543,24.790,154.513
C06311=1068.511,-0.667,-64.365,172.544,24.793,154.513
C06312=1068.517,-0.418,-64.379,172.545,24.796,154.514
C06313=1068.523,-0.167,-64.394,172.547,24.798,154.514
C06314=1068.530,0.081,-64.408,172.548,24.800,154.514
C06315=1068.536,0.332,-64.422,172.550,24.803,154.515
C06316=1068.542,0.581,-64.436,172.551,24.806,154.515
C06317=1068.547,0.830,-64.450,172.552,24.808,154.515
C06318=1068.554,1.080,-64.465,172.554,24.810,154.515
C06319=1068.559,1.329,-64.479,172.555,24.813,154.516
C06320=1068.565,1.579,-64.494,172.556,24.816,154.516
C06321=1068.571,1.829,-64.508,172.558,24.818,154.516
C06322=1068.577,2.078,-64.522,172.559,24.820,154.517
C06323=1068.583,2.327,-64.537,172.561,24.823,154.517
C06324=1068.589,2.577,-64.551,172.562,24.826,154.517
C06325=1068.595,2.826,-64.566,172.563,24.828,154.518
C06326=1068.600,3.076,-64.580,172.565,24.830,154.518
C06327=1068.607,3.326,-64.595,172.566,24.833,154.518
C06328=1068.612,3.575,-64.609,172.567,24.836,154.519
C06329=1068.619,3.825,-64.624,172.570,24.838,154.519
C06330=1068.624,4.074,-64.638,172.571,24.841,154.519
C06331=1068.630,4.323,-64.652,172.572,24.844,154.520
C06332=1068.636,4.573,-64.667,172.574,24.846,154.520
C06333=1068.642,4.822,-64.682,172.575,24.848,154.520
C06334=1068.648,5.072,-64.696,172.577,24.851,154.520
C06335=1068.654,5.321,-64.711,172.578,24.854,154.521
C06336=1068.660,5.571,-64.726,172.579,24.856,154.521
C06337=1068.666,5.821,-64.739,172.581,24.858,154.521
C06338=1068.672,6.070,-64.754,172.582,24.861,154.522
C06339=1068.678,6.319,-64.769,172.583,24.864,154.522
C06340=1068.684,6.569,-64.783,172.585,24.866,154.522
C06341=1068.690,6.818,-64.798,172.586,24.868,154.523
C06342=1068.696,7.068,-64.813,172.587,24.871,154.523
C06343=1068.702,7.318,-64.827,172.589,24.874,154.523
C06344=1068.708,7.567,-64.842,172.590,24.876,154.523
C06345=1068.714,7.817,-64.856,172.591,24.879,154.524
C06346=1068.720,8.066,-64.871,172.593,24.881,154.524
C06347=1068.726,8.316,-64.885,172.594,24.884,154.524
C06348=1068.732,8.565,-64.900,172.596,24.886,154.525
C06349=1068.738,8.815,-64.915,172.597,24.889,154.525
C06350=1068.744,9.064,-64.929,172.598,24.891,154.525
C06351=1068.750,9.314,-64.944,172.600,24.894,154.526
C06352=1068.756,9.563,-64.958,172.601,24.897,154.526
C06353=1068.762,9.813,-64.973,172.602,24.899,154.526
C06354=1068.769,10.062,-64.988,172.604,24.901,154.527
C06355=1068.775,10.311,-65.003,172.605,24.904,154.527
C06356=1068.781,10.561,-65.017,172.607,24.907,154.527
C06357=1068.786,10.810,-65.031,172.608,24.909,154.528
C06358=1068.793,11.060,-65.046,172.609,24.911,154.528
C06359=1068.799,11.309,-65.061,172.611,24.914,154.528
C06360=1068.804,11.559,-65.077,172.612,24.917,154.528
C06361=1068.811,11.809,-65.091,172.614,24.919,154.529
C06362=1068.816,12.058,-65.105,172.616,24.922,154.529
C06363=1068.823,12.308,-65.120,172.617,24.925,154.529
C06364=1068.829,12.558,-65.135,172.619,24.927,154.530
C06365=1068.835,12.807,-65.150,172.620,24.929,154.530
C06366=1068.841,13.056,-65.165,172.621,24.932,154.530
C06367=1068.847,13.305,-65.179,172.623,24.935,154.531
C06368=1068.853,13.555,-65.194,172.624,24.937,154.531
C06369=1068.860,13.804,-65.209,172.625,24.939,154.531
C06370=1068.866,14.086,-65.226,172.627,24.942,154.532
C06371=1068.873,14.367,-65.243,172.628,24.945,154.532
C06372=1068.879,14.649,-65.259,172.630,24.948,154.532
C06373=1068.886,14.931,-65.276,172.632,24.951,154.533
C06374=1068.892,15.181,-65.291,172.633,24.954,154.533
C06375=1068.898,15.430,-65.306,172.634,24.956,154.533
C06376=1068.904,15.679,-65.321,172.636,24.959,154.534
C06377=1068.909,15.928,-65.336,172.637,24.961,154.534
C06378=1068.916,16.178,-65.351,172.638,24.964,154.534
C06379=1068.922,16.428,-65.366,172.640,24.967,154.535
C06380=1068.927,16.677,-65.381,172.641,24.969,154.535
C06381=1068.934,16.927,-65.396,172.642,24.972,154.535
C06382=1068.940,17.176,-65.411,172.644,24.974,154.536
C06383=1068.945,17.426,-65.426,172.645,24.977,154.536
C06384=1068.951,17.675,-65.441,172.646,24.980,154.536
C06385=1068.958,17.924,-65.456,172.648,24.982,154.537
C06386=1068.964,18.173,-65.471,172.649,24.985,154.537
C06387=1068.970,18.423,-65.487,172.651,24.987,154.537
C06388=1068.976,18.673,-65.501,172.652,24.990,154.537
C06389=1068.982,18.922,-65.516,172.653,24.992,154.538
C06390=1068.987,19.172,-65.532,172.655,24.995,154.538
C06391=1068.994,19.421,-65.547,172.656,24.998,154.539
C06392=1069.000,19.670,-65.561,172.657,25.000,154.539
C06393=1069.005,19.920,-65.577,172.659,25.002,154.539
C06394=1069.012,20.170,-65.592,172.660,25.005,154.540
C06395=1069.017,20.419,-65.606,172.661,25.008,154.540
C06396=1069.023,20.668,-65.622,172.664,25.011,154.540
C06397=1069.030,20.918,-65.637,172.665,25.013,154.540
C06398=1069.035,21.167,-65.653,172.666,25.016,154.541
C06399=1069.041,21.417,-65.668,172.668,25.019,154.541
C06400=1069.047,21.667,-65.683,172.669,25.021,154.541
C06401=1069.053,21.916,-65.698,172.671,25.024,154.542
C06402=1069.059,22.165,-65.713,172.672,25.026,154.542
C06403=1069.065,22.415,-65.729,172.673,25.029,154.542
C06404=1069.071,22.665,-65.744,172.675,25.031,154.543
C06405=1069.076,22.914,-65.759,172.676,25.034,154.543
C06406=1069.083,23.163,-65.774,172.677,25.037,154.543
C06407=1069.089,23.413,-65.790,172.679,25.040,154.544
C06408=1069.094,23.662,-65.805,172.680,25.042,154.544
C06409=1069.100,23.912,-65.820,172.681,25.044,154.544
C06410=1069.106,24.161,-65.835,172.683,25.047,154.545
C06411=1069.113,24.410,-65.851,172.684,25.050,154.545
C06412=1069.118,24.660,-65.866,172.685,25.052,154.545
C06413=1069.125,24.909,-65.881,172.687,25.055,154.546
C06414=1069.130,25.159,-65.897,172.688,25.058,154.546
C06415=1069.137,25.408,-65.912,172.690,25.060,154.546
C06416=1069.142,25.658,-65.927,172.691,25.063,154.547
C06417=1069.148,25.907,-65.942,172.692,25.065,154.547
C06418=1069.154,26.157,-65.958,172.694,25.068,154.547
C06419=1069.161,26.406,-65.974,172.695,25.071,154.548
C06420=1069.166,26.656,-65.989,172.696,25.073,154.548
C06421=1069.172,26.905,-66.004,172.698,25.076,154.548
C06422=1069.178,27.155,-66.020,172.699,25.078,154.549
C06423=1069.184,27.404,-66.035,172.700,25.081,154.549
C06424=1069.190,27.654,-66.050,172.702,25.083,154.549
C06425=1069.196,27.903,-66.066,172.703,25.086,154.550
C06426=1069.202,28.152,-66.081,172.705,25.089,154.550
C06427=1069.208,28.402,-66.098,172.706,25.092,154.550
C06428=1069.214,28.651,-66.112,172.707,25.094,154.551
C06429=1069.219,28.901,-66.128,172.709,25.097,154.551
C06430=1069.226,29.150,-66.143,172.711,25.100,154.551
C06431=1069.232,29.400,-66.159,172.712,25.102,154.552
C06432=1069.237,29.649,-66.175,172.714,25.105,154.552
C06433=1069.244,29.899,-66.190,172.715,25.108,154.552
C06434=1069.250,30.181,-66.207,172.716,25.111,154.553
C06435=1069.257,30.464,-66.225,172.717,25.114,154.553
C06436=1069.264,30.747,-66.243,172.720,25.117,154.554
C06437=1069.270,31.030,-66.261,172.721,25.120,154.554
C06438=1069.276,31.280,-66.277,172.722,25.122,154.554
C06439=1069.282,31.528,-66.292,172.724,25.125,154.555
C06440=1069.288,31.778,-66.307,172.725,25.127,154.555
C06441=1069.293,32.028,-66.324,172.726,25.130,154.555
C06442=1069.300,32.277,-66.339,172.728,25.133,154.556
C06443=1069.306,32.527,-66.355,172.729,25.135,154.556
C06444=1069.311,32.777,-66.370,172.731,25.138,154.556
C06445=1069.318,33.025,-66.386,172.732,25.141,154.557
C06446=1069.323,33.275,-66.401,172.733,25.143,154.557
C06447=1069.329,33.524,-66.417,172.735,25.146,154.557
C06448=1069.335,33.774,-66.434,172.736,25.148,154.558
C06449=1069.341,34.023,-66.449,172.737,25.151,154.558
C06450=1069.347,34.273,-66.465,172.739,25.154,154.558
C06451=1069.353,34.523,-66.480,172.740,25.156,154.559
C06452=1069.359,34.771,-66.496,172.741,25.159,154.559
C06453=1069.365,35.021,-66.511,172.743,25.162,154.559
C06454=1069.371,35.270,-66.528,172.744,25.164,154.560
C06455=1069.377,35.520,-66.544,172.745,25.167,154.560
C06456=1069.383,35.769,-66.559,172.747,25.169,154.560
C06457=1069.389,36.019,-66.575,172.748,25.172,154.561
C06458=1069.395,36.269,-66.591,172.750,25.175,154.561
C06459=1069.401,36.518,-66.607,172.752,25.178,154.561
C06460=1069.407,36.767,-66.623,172.753,25.180,154.562
C06461=1069.413,37.017,-66.638,172.755,25.183,154.562
C06462=1069.418,37.266,-66.654,172.756,25.185,154.562
C06463=1069.424,37.515,-66.670,172.757,25.188,154.563
C06464=1069.431,37.765,-66.685,172.759,25.191,154.563
C06465=1069.437,38.014,-66.701,172.760,25.193,154.563
C06466=1069.443,38.263,-66.718,172.761,25.196,154.564
C06467=1069.448,38.513,-66.733,172.763,25.199,154.564
C06468=1069.454,38.763,-66.749,172.764,25.202,154.565
C06469=1069.460,39.012,-66.766,172.765,25.204,154.565
C06470=1069.466,39.261,-66.782,172.767,25.207,154.565
C06471=1069.472,39.511,-66.798,172.768,25.210,154.566
C06472=1069.477,39.760,-66.813,172.769,25.212,154.566
C06473=1069.483,40.009,-66.830,172.771,25.215,154.566
C06474=1069.490,40.258,-66.845,172.772,25.217,154.567
C06475=1069.495,40.508,-66.861,172.773,25.220,154.567
C06476=1069.501,40.758,-66.877,172.775,25.223,154.567
C06477=1069.507,41.007,-66.893,172.776,25.225,154.568
C06478=1069.513,41.256,-66.910,172.778,25.228,154.568
C06479=1069.519,41.506,-66.926,172.779,25.231,154.568
C06480=1069.525,41.756,-66.941,172.780,25.234,154.569
C06481=1069.531,42.005,-66.958,172.782,25.236,154.569
C06482=1069.537,42.254,-66.974,172.783,25.239,154.569
C06483=1069.543,42.504,-66.990,172.784,25.241,154.570
C06484=1069.549,42.753,-67.006,172.786,25.244,154.570
C06485=1069.554,43.003,-67.022,172.788,25.247,154.570
C06486=1069.560,43.252,-67.038,172.789,25.250,154.571
C06487=1069.566,43.502,-67.054,172.791,25.253,154.571
C06488=1069.572,43.751,-67.071,172.792,25.255,154.571
C06489=1069.577,44.000,-67.087,172.793,25.258,154.572
C06490=1069.583,44.249,-67.103,172.795,25.261,154.572
C06491=1069.589,44.498,-67.119,172.796,25.263,154.573
C06492=1069.595,44.748,-67.135,172.797,25.266,154.573
C06493=1069.601,44.997,-67.152,172.799,25.269,154.573
C06494=1069.606,45.247,-67.168,172.800,25.271,154.574
C06495=1069.612,45.497,-67.184,172.801,25.274,154.574
C06496=1069.618,45.746,-67.200,172.803,25.277,154.574
C06497=1069.624,45.995,-67.217,172.804,25.279,154.575
C06498=1069.630,46.278,-67.236,172.806,25.282,154.575
C06499=1069.637,46.561,-67.254,172.808,25.286,154.576
C06500=1069.643,46.844,-67.273,172.809,25.289,154.576
C06501=1069.650,47.127,-67.291,172.810,25.292,154.576
C06502=1069.656,47.376,-67.307,172.812,25.295,154.577
C06503=1069.662,47.626,-67.323,172.813,25.297,154.577
C06504=1069.667,47.875,-67.340,172.814,25.300,154.577
C06505=1069.673,48.125,-67.356,172.816,25.303,154.578
C06506=1069.679,48.374,-67.372,172.817,25.305,154.578
C06507=1069.685,48.623,-67.389,172.818,25.308,154.579
C06508=1069.691,48.873,-67.405,172.821,25.311,154.579
C06509=1069.696,49.122,-67.422,172.822,25.313,154.579
C06510=1069.702,49.371,-67.439,172.823,25.316,154.580
C06511=1069.708,49.620,-67.455,172.825,25.319,154.580
C06512=1069.714,49.870,-67.471,172.826,25.322,154.580
C06513=1069.720,50.119,-67.488,172.827,25.324,154.581
C06514=1069.725,50.369,-67.504,172.829,25.327,154.581
C06515=1069.731,50.618,-67.521,172.830,25.330,154.581
C06516=1069.737,50.867,-67.537,172.831,25.333,154.582
C06517=1069.743,51.117,-67.553,172.833,25.335,154.582
C06518=1069.749,51.366,-67.570,172.834,25.338,154.582
C06519=1069.755,51.616,-67.587,172.836,25.340,154.583
C06520=1069.761,51.866,-67.603,172.837,25.343,154.583
C06521=1069.767,52.115,-67.620,172.838,25.346,154.584
C06522=1069.773,52.364,-67.637,172.840,25.348,154.584
C06523=1069.778,52.614,-67.653,172.841,25.351,154.584
C06524=1069.784,52.863,-67.669,172.842,25.354,154.585
C06525=1069.790,53.112,-67.685,172.844,25.356,154.585
C06526=1069.796,53.362,-67.702,172.845,25.359,154.585
C06527=1069.802,53.611,-67.719,172.846,25.362,154.586
C06528=1069.808,53.860,-67.736,172.848,25.364,154.586
C06529=1069.814,54.109,-67.752,172.850,25.368,154.586
C06530=1069.819,54.359,-67.769,172.851,25.370,154.587
C06531=1069.826,54.609,-67.785,172.853,25.373,154.587
C06532=1069.832,54.858,-67.802,172.854,25.375,154.587
C06533=1069.838,55.107,-67.819,172.856,25.378,154.588
C06534=1069.843,55.357,-67.835,172.857,25.381,154.588
C06535=1069.849,55.606,-67.852,172.858,25.383,154.588
C06536=1069.855,55.855,-67.869,172.860,25.386,154.589
C06537=1069.861,56.104,-67.885,172.861,25.389,154.589
C06538=1069.867,56.355,-67.902,172.862,25.391,154.589
C06539=1069.873,56.604,-67.918,172.864,25.394,154.590
C06540=1069.879,56.853,-67.935,172.865,25.397,154.590
C06541=1069.884,57.102,-67.952,172.866,25.400,154.591
C06542=1069.890,57.352,-67.968,172.868,25.402,154.591
C06543=1069.897,57.600,-67.985,172.869,25.405,154.591
C06544=1069.903,57.850,-68.002,172.871,25.407,154.592
C06545=1069.908,58.100,-68.019,172.872,25.410,154.592
C06546=1069.915,58.349,-68.036,172.873,25.413,154.592
C06547=1069.921,58.598,-68.052,172.876,25.416,154.593
C06548=1069.926,58.848,-68.069,172.877,25.418,154.593
C06549=1069.933,59.097,-68.086,172.878,25.421,154.593
C06550=1069.939,59.347,-68.103,172.880,25.424,154.594
C06551=1069.944,59.596,-68.119,172.881,25.426,154.594
C06552=1069.950,59.845,-68.136,172.882,25.429,154.594
C06553=1069.956,60.094,-68.153,172.884,25.432,154.595
C06554=1069.962,60.344,-68.171,172.885,25.434,154.595
C06555=1069.968,60.593,-68.187,172.887,25.437,154.595
C06556=1069.974,60.843,-68.203,172.888,25.439,154.596
C06557=1069.979,61.092,-68.221,172.889,25.442,154.596
C06558=1069.986,61.342,-68.237,172.891,25.444,154.596
C06559=1069.992,61.591,-68.254,172.892,25.447,154.597
C06560=1069.998,61.840,-68.271,172.894,25.450,154.597
C06561=1070.004,62.089,-68.288,172.895,25.453,154.597
C06562=1070.011,62.372,-68.307,172.897,25.456,154.598
C06563=1070.018,62.654,-68.326,172.898,25.459,154.598
C06564=1070.024,62.937,-68.345,172.900,25.461,154.599
C06565=1070.031,63.219,-68.365,172.902,25.465,154.599
C06566=1070.037,63.470,-68.382,172.903,25.467,154.599
C06567=1070.043,63.718,-68.399,172.905,25.470,154.600
C06568=1070.049,63.968,-68.415,172.906,25.473,154.600
C06569=1070.055,64.217,-68.433,172.908,25.475,154.600
C06570=1070.061,64.467,-68.449,172.909,25.478,154.601
C06571=1070.067,64.716,-68.467,172.910,25.480,154.601
C06572=1070.073,64.965,-68.483,172.912,25.483,154.601
C06573=1070.079,65.215,-68.501,172.913,25.485,154.602
C06574=1070.085,65.464,-68.517,172.914,25.488,154.602
C06575=1070.090,65.713,-68.535,172.916,25.491,154.603
C06576=1070.096,65.963,-68.552,172.918,25.494,154.603
C06577=1070.103,66.212,-68.569,172.919,25.497,154.603
C06578=1070.108,66.461,-68.587,172.921,25.500,154.604
C06579=1070.114,66.711,-68.603,172.922,25.502,154.604
C06580=1070.120,66.960,-68.620,172.924,25.505,154.604
C06581=1070.126,67.209,-68.638,172.925,25.507,154.605
C06582=1070.132,67.459,-68.655,172.926,25.510,154.605
C06583=1070.137,67.708,-68.672,172.928,25.513,154.605
C06584=1070.144,67.958,-68.689,172.929,25.515,154.606
C06585=1070.149,68.207,-68.706,172.930,25.518,154.606
C06586=1070.155,68.456,-68.724,172.932,25.521,154.606
C06587=1070.161,68.705,-68.740,172.933,25.523,154.607
C06588=1070.167,68.955,-68.758,172.935,25.526,154.607
C06589=1070.172,69.204,-68.776,172.936,25.529,154.607
C06590=1070.179,69.453,-68.793,172.938,25.532,154.608
C06591=1070.184,69.703,-68.810,172.940,25.535,154.608
C06592=1070.191,69.952,-68.827,172.941,25.537,154.608
C06593=1070.196,70.201,-68.844,172.942,25.540,154.609
C06594=1070.202,70.451,-68.862,172.944,25.543,154.609
C06595=1070.207,70.700,-68.879,172.945,25.545,154.610
C06596=1070.214,70.949,-68.896,172.946,25.548,154.610
C06597=1070.220,71.199,-68.914,172.948,25.551,154.610
C06598=1070.225,71.449,-68.931,172.949,25.553,154.611
C06599=1070.231,71.698,-68.948,172.951,25.556,154.611
C06600=1070.237,71.947,-68.966,172.952,25.559,154.611
C06601=1070.243,72.196,-68.983,172.953,25.561,154.612
C06602=1070.248,72.445,-69.001,172.955,25.564,154.612
C06603=1070.254,72.695,-69.018,172.957,25.567,154.612
C06604=1070.260,72.945,-69.036,172.958,25.569,154.613
C06605=1070.266,73.193,-69.053,172.960,25.572,154.613
C06606=1070.272,73.443,-69.071,172.961,25.575,154.613
C06607=1070.278,73.692,-69.088,172.963,25.578,154.614
C06608=1070.283,73.941,-69.106,172.964,25.580,154.614
C06609=1070.289,74.191,-69.123,172.965,25.583,154.615
C06610=1070.295,74.440,-69.140,172.967,25.586,154.615
C06611=1070.301,74.689,-69.157,172.968,25.588,154.615
C06612=1070.307,74.939,-69.175,172.969,25.591,154.616
C06613=1070.312,75.188,-69.193,172.971,25.594,154.616
C06614=1070.319,75.438,-69.211,172.972,25.597,154.616
C06615=1070.325,75.686,-69.228,172.974,25.599,154.617
C06616=1070.330,75.935,-69.245,172.976,25.602,154.617
C06617=1070.336,76.185,-69.263,172.977,25.604,154.617
C06618=1070.342,76.434,-69.281,172.979,25.607,154.618
C06619=1070.348,76.685,-69.298,172.980,25.610,154.618
C06620=1070.354,76.933,-69.315,172.981,25.612,154.618
C06621=1070.360,77.182,-69.333,172.983,25.615,154.619
C06622=1070.366,77.432,-69.351,172.984,25.618,154.619
C06623=1070.371,77.681,-69.368,172.986,25.620,154.620
C06624=1070.377,77.931,-69.386,172.987,25.623,154.620
C06625=1070.383,78.180,-69.404,172.988,25.626,154.620
C06626=1070.389,78.462,-69.423,172.991,25.629,154.621
C06627=1070.397,78.744,-69.444,172.992,25.632,154.621
C06628=1070.403,79.027,-69.464,172.994,25.635,154.622
C06629=1070.409,79.309,-69.484,172.995,25.638,154.622
C06630=1070.415,79.559,-69.502,172.997,25.641,154.622
C06631=1070.421,79.808,-69.520,172.998,25.643,154.623
C06632=1070.427,80.058,-69.538,173.000,25.646,154.623
C06633=1070.432,80.307,-69.555,173.001,25.649,154.623
C06634=1070.439,80.557,-69.573,173.002,25.652,154.624
C06635=1070.444,80.806,-69.591,173.005,25.655,154.624
C06636=1070.450,81.055,-69.608,173.006,25.658,154.624
C06637=1070.456,81.304,-69.626,173.007,25.660,154.625
C06638=1070.461,81.553,-69.644,173.009,25.663,154.625
C06639=1070.468,81.803,-69.662,173.010,25.666,154.626
C06640=1070.473,82.052,-69.680,173.012,25.668,154.626
C06641=1070.479,82.301,-69.698,173.013,25.671,154.626
C06642=1070.484,82.551,-69.716,173.014,25.674,154.627
C06643=1070.490,82.800,-69.734,173.016,25.676,154.627
C06644=1070.496,83.049,-69.752,173.017,25.679,154.627
C06645=1070.501,83.299,-69.769,173.019,25.682,154.628
C06646=1070.508,83.548,-69.788,173.021,25.684,154.628
C06647=1070.513,83.797,-69.805,173.022,25.687,154.628
C06648=1070.519,84.046,-69.823,173.023,25.690,154.629
C06649=1070.525,84.295,-69.841,173.025,25.692,154.629
C06650=1070.531,84.545,-69.859,173.026,25.695,154.629
C06651=1070.537,84.794,-69.877,173.028,25.698,154.630
C06652=1070.543,85.043,-69.895,173.029,25.700,154.630
C06653=1070.548,85.292,-69.913,173.030,25.703,154.631
C06654=1070.554,85.542,-69.931,173.033,25.706,154.631
C06655=1070.560,85.791,-69.949,173.034,25.709,154.631
C06656=1070.566,86.041,-69.967,173.035,25.712,154.632
C06657=1070.571,86.290,-69.985,173.037,25.714,154.632
C06658=1070.577,86.539,-70.003,173.038,25.717,154.632
C06659=1070.584,86.789,-70.021,173.040,25.720,154.633
C06660=1070.589,87.038,-70.039,173.041,25.722,154.633
C06661=1070.595,87.287,-70.057,173.042,25.725,154.633
C06662=1070.601,87.536,-70.074,173.044,25.727,154.634
C06663=1070.607,87.786,-70.094,173.046,25.730,154.634
C06664=1070.612,88.035,-70.111,173.048,25.733,154.634
C06665=1070.618,88.285,-70.129,173.049,25.735,154.635
C06666=1070.624,88.533,-70.147,173.050,25.738,154.635
C06667=1070.630,88.783,-70.165,173.052,25.741,154.635
C06668=1070.636,89.032,-70.183,173.053,25.743,154.636
C06669=1070.642,89.281,-70.202,173.055,25.746,154.636
C06670=1070.648,89.531,-70.220,173.056,25.749,154.637
C06671=1070.653,89.779,-70.238,173.058,25.752,154.637
C06672=1070.659,90.029,-70.256,173.060,25.754,154.637
C06673=1070.666,90.279,-70.274,173.061,25.757,154.638
C06674=1070.671,90.527,-70.293,173.063,25.759,154.638
C06675=1070.678,90.777,-70.311,173.064,25.762,154.638
C06676=1070.683,91.026,-70.329,173.065,25.765,154.639
C06677=1070.689,91.275,-70.347,173.067,25.767,154.639
C06678=1070.695,91.525,-70.365,173.068,25.770,154.639
C06679=1070.700,91.774,-70.384,173.070,25.773,154.640
C06680=1070.706,92.024,-70.402,173.072,25.776,154.640
C06681=1070.712,92.272,-70.420,173.073,25.778,154.640
C06682=1070.717,92.522,-70.439,173.074,25.781,154.641
C06683=1070.723,92.771,-70.457,173.076,25.784,154.641
C06684=1070.729,93.020,-70.475,173.077,25.786,154.642
C06685=1070.735,93.270,-70.494,173.079,25.789,154.642
C06686=1070.740,93.519,-70.512,173.080,25.792,154.642
C06687=1070.746,93.768,-70.531,173.082,25.795,154.643
C06688=1070.752,94.017,-70.549,173.084,25.798,154.643
C06689=1070.758,94.266,-70.567,173.085,25.800,154.643
C06690=1070.765,94.549,-70.589,173.087,25.803,154.644
C06691=1070.771,94.832,-70.609,173.089,25.806,154.644
C06692=1070.777,95.114,-70.630,173.090,25.809,154.645
C06693=1070.784,95.397,-70.652,173.092,25.813,154.645
C06694=1070.789,95.646,-70.669,173.094,25.815,154.645
C06695=1070.796,95.895,-70.688,173.095,25.818,154.646
C06696=1070.801,96.145,-70.707,173.097,25.821,154.646
C06697=1070.807,96.393,-70.725,173.098,25.823,154.646
C06698=1070.813,96.643,-70.744,173.099,25.826,154.647
C06699=1070.819,96.893,-70.762,173.101,25.828,154.647
C06700=1070.825,97.141,-70.780,173.103,25.831,154.647
C06701=1070.830,97.390,-70.799,173.104,25.834,154.648
C06702=1070.836,97.640,-70.817,173.106,25.836,154.648
C06703=1070.842,97.889,-70.836,173.107,25.839,154.648
C06704=1070.848,98.138,-70.855,173.109,25.841,154.649
C06705=1070.854,98.388,-70.873,173.110,25.844,154.649
C06706=1070.859,98.637,-70.892,173.112,25.847,154.650
C06707=1070.866,98.886,-70.910,173.114,25.850,154.650
C06708=1070.871,99.136,-70.929,173.115,25.853,154.650
C06709=1070.877,99.384,-70.947,173.117,25.855,154.651
C06710=1070.883,99.634,-70.966,173.118,25.858,154.651
C06711=1070.889,99.883,-70.984,173.120,25.860,154.651
C06712=1070.894,100.133,-71.004,173.121,25.863,154.652
C06713=1070.900,100.381,-71.022,173.123,25.866,154.652
C06714=1070.907,100.630,-71.041,173.125,25.868,154.652
C06715=1070.912,100.880,-71.059,173.126,25.871,154.653
C06716=1070.918,101.129,-71.078,173.128,25.874,154.653
C06717=1070.923,101.378,-71.097,173.129,25.876,154.653
C06718=1070.929,101.628,-71.116,173.130,25.879,154.654
C06719=1070.936,101.877,-71.135,173.133,25.882,154.654
C06720=1070.940,102.126,-71.153,173.134,25.885,154.654
C06721=1070.946,102.376,-71.172,173.135,25.888,154.655
C06722=1070.952,102.625,-71.191,173.137,25.890,154.655
C06723=1070.958,102.874,-71.210,173.138,25.893,154.656
C06724=1070.963,103.123,-71.229,173.140,25.896,154.656
C06725=1070.970,103.372,-71.247,173.141,25.898,154.656
C06726=1070.975,103.622,-71.266,173.143,25.901,154.657
C06727=1070.980,103.871,-71.285,173.145,25.904,154.657
C06728=1070.987,104.120,-71.303,173.146,25.906,154.657
C06729=1070.992,104.369,-71.323,173.148,25.909,154.658
C06730=1070.998,104.619,-71.342,173.149,25.911,154.658
C06731=1071.004,104.867,-71.360,173.151,25.914,154.658
C06732=1071.009,105.117,-71.379,173.153,25.917,154.659
C06733=1071.015,105.366,-71.399,173.154,25.920,154.659
C06734=1071.022,105.615,-71.417,173.156,25.922,154.659
C06735=1071.027,105.864,-71.436,173.157,25.925,154.660
C06736=1071.032,106.114,-71.455,173.158,25.928,154.660
C06737=1071.038,106.363,-71.473,173.161,25.931,154.661
C06738=1071.044,106.612,-71.493,173.162,25.933,154.661
C06739=1071.050,106.862,-71.512,173.164,25.936,154.661
C06740=1071.055,107.111,-71.531,173.165,25.939,154.662
C06741=1071.061,107.360,-71.549,173.166,25.941,154.662
C06742=1071.067,107.609,-71.569,173.168,25.944,154.662
C06743=1071.073,107.859,-71.588,173.170,25.946,154.663
C06744=1071.079,108.108,-71.606,173.172,25.949,154.663
C06745=1071.084,108.356,-71.625,173.173,25.952,154.663
C06746=1071.090,108.606,-71.645,173.174,25.954,154.664
C06747=1071.096,108.855,-71.664,173.176,25.957,154.664
C06748=1071.102,109.104,-71.683,173.178,25.960,154.664
C06749=1071.108,109.353,-71.702,173.180,25.963,154.665
C06750=1071.114,109.603,-71.722,173.181,25.965,154.665
C06751=1071.120,109.851,-71.740,173.182,25.968,154.665
C06752=1071.125,110.101,-71.759,173.184,25.971,154.666
C06753=1071.131,110.350,-71.778,173.186,25.973,154.666
C06754=1071.138,110.633,-71.800,173.188,25.976,154.666
C06755=1071.144,110.915,-71.821,173.190,25.979,154.667
C06756=1071.151,111.198,-71.844,173.191,25.982,154.667
C06757=1071.157,111.480,-71.865,173.193,25.985,154.668
C06758=1071.163,111.730,-71.884,173.195,25.988,154.668
C06759=1071.169,111.979,-71.904,173.196,25.990,154.668
C06760=1071.174,112.228,-71.923,173.198,25.993,154.669
C06761=1071.181,112.478,-71.942,173.199,25.996,154.669
C06762=1071.187,112.726,-71.962,173.201,25.998,154.669
C06763=1071.192,112.976,-71.981,173.203,26.001,154.670
C06764=1071.198,113.225,-72.000,173.204,26.004,154.670
C06765=1071.203,113.474,-72.019,173.206,26.007,154.670
C06766=1071.209,113.723,-72.038,173.207,26.009,154.671
C06767=1071.215,113.972,-72.058,173.210,26.012,154.671
C06768=1071.221,114.222,-72.077,173.211,26.015,154.672
C06769=1071.226,114.471,-72.097,173.212,26.017,154.672
C06770=1071.232,114.721,-72.116,173.214,26.020,154.672
C06771=1071.238,114.969,-72.136,173.215,26.023,154.673
C06772=1071.243,115.218,-72.155,173.218,26.025,154.673
C06773=1071.249,115.467,-72.174,173.219,26.028,154.673
C06774=1071.255,115.716,-72.194,173.220,26.031,154.674
C06775=1071.260,115.966,-72.213,173.222,26.033,154.674
C06776=1071.266,116.215,-72.232,173.223,26.036,154.674
C06777=1071.272,116.465,-72.252,173.225,26.039,154.675
C06778=1071.278,116.713,-72.272,173.227,26.042,154.675
C06779=1071.283,116.962,-72.290,173.228,26.045,154.675
C06780=1071.288,117.212,-72.310,173.230,26.047,154.676
C06781=1071.294,117.461,-72.330,173.231,26.050,154.676
C06782=1071.299,117.710,-72.350,173.233,26.053,154.677
C06783=1071.305,117.959,-72.369,173.235,26.056,154.677
C06784=1071.311,118.208,-72.389,173.236,26.058,154.677
C06785=1071.317,118.458,-72.408,173.238,26.061,154.678
C06786=1071.323,118.707,-72.428,173.240,26.064,154.678
C06787=1071.329,118.956,-72.447,173.242,26.066,154.678
C06788=1071.334,119.205,-72.468,173.243,26.069,154.679
C06789=1071.339,119.455,-72.487,173.244,26.072,154.679
C06790=1071.345,119.703,-72.506,173.246,26.074,154.679
C06791=1071.351,119.952,-72.526,173.248,26.077,154.680
C06792=1071.356,120.202,-72.545,173.250,26.080,154.680
C06793=1071.362,120.450,-72.565,173.251,26.082,154.680
C06794=1071.368,120.700,-72.584,173.252,26.085,154.681
C06795=1071.374,120.949,-72.604,173.255,26.088,154.681
C06796=1071.379,121.198,-72.624,173.256,26.091,154.682
C06797=1071.385,121.447,-72.644,173.258,26.093,154.682
C06798=1071.391,121.697,-72.663,173.259,26.096,154.682
C06799=1071.397,121.945,-72.683,173.261,26.099,154.683
C06800=1071.402,122.195,-72.702,173.263,26.101,154.683
C06801=1071.408,122.444,-72.722,173.264,26.104,154.683
C06802=1071.413,122.693,-72.742,173.266,26.106,154.684
C06803=1071.419,122.942,-72.762,173.268,26.109,154.684
C06804=1071.425,123.192,-72.781,173.269,26.112,154.684
C06805=1071.431,123.441,-72.801,173.271,26.114,154.685
C06806=1071.437,123.689,-72.821,173.272,26.117,154.685
C06807=1071.442,123.939,-72.841,173.275,26.120,154.685
C06808=1071.448,124.188,-72.861,173.276,26.123,154.686
C06809=1071.453,124.437,-72.880,173.278,26.125,154.686
C06810=1071.459,124.686,-72.900,173.279,26.128,154.686
C06811=1071.465,124.935,-72.920,173.281,26.131,154.687
C06812=1071.471,125.184,-72.940,173.283,26.133,154.687
C06813=1071.477,125.434,-72.960,173.284,26.136,154.687
C06814=1071.483,125.684,-72.980,173.286,26.138,154.688
C06815=1071.489,125.932,-73.000,173.288,26.142,154.688
C06816=1071.495,126.181,-73.020,173.289,26.144,154.688
C06817=1071.500,126.431,-73.039,173.291,26.147,154.689
C06818=1071.507,126.713,-73.062,173.293,26.150,154.689
C06819=1071.513,126.995,-73.084,173.295,26.153,154.690
C06820=1071.520,127.278,-73.107,173.297,26.156,154.690
C06821=1071.526,127.561,-73.130,173.298,26.159,154.690
C06822=1071.532,127.809,-73.150,173.301,26.161,154.691
C06823=1071.538,128.059,-73.169,173.302,26.164,154.691
C06824=1071.544,128.308,-73.189,173.304,26.166,154.691
C06825=1071.549,128.557,-73.210,173.306,26.169,154.692
C06826=1071.556,128.806,-73.230,173.307,26.172,154.692
C06827=1071.561,129.056,-73.249,173.309,26.174,154.692
C06828=1071.567,129.305,-73.269,173.310,26.177,154.693
C06829=1071.572,129.554,-73.290,173.313,26.180,154.693
C06830=1071.578,129.803,-73.310,173.314,26.182,154.693
C06831=1071.584,130.051,-73.330,173.315,26.185,154.694
C06832=1071.591,130.301,-73.349,173.318,26.188,154.694
C06833=1071.596,130.551,-73.370,173.319,26.190,154.694
C06834=1071.602,130.799,-73.390,173.321,26.193,154.695
C06835=1071.608,131.048,-73.410,173.322,26.195,154.695
C06836=1071.614,131.297,-73.430,173.325,26.198,154.695
C06837=1071.619,131.546,-73.450,173.326,26.201,154.696
C06838=1071.626,131.796,-73.470,173.327,26.203,154.696
C06839=1071.632,132.045,-73.490,173.330,26.206,154.696
C06840=1071.637,132.294,-73.510,173.331,26.209,154.697
C06841=1071.643,132.543,-73.530,173.333,26.211,154.697
C06842=1071.648,132.792,-73.551,173.334,26.214,154.697
C06843=1071.654,133.041,-73.571,173.337,26.217,154.698
C06844=1071.659,133.290,-73.591,173.338,26.219,154.698
C06845=1071.666,133.540,-73.612,173.339,26.222,154.698
C06846=1071.671,133.789,-73.632,173.342,26.225,154.699
C06847=1071.677,134.038,-73.652,173.343,26.227,154.699
C06848=1071.682,134.287,-73.673,173.345,26.230,154.700
C06849=1071.688,134.535,-73.693,173.347,26.233,154.700
C06850=1071.694,134.785,-73.713,173.348,26.235,154.700
C06851=1071.700,135.034,-73.734,173.350,26.238,154.701
C06852=1071.705,135.283,-73.754,173.351,26.241,154.701
C06853=1071.711,135.532,-73.774,173.354,26.244,154.701
C06854=1071.717,135.781,-73.795,173.355,26.246,154.702
C06855=1071.723,136.030,-73.815,173.357,26.249,154.702
C06856=1071.729,136.280,-73.836,173.359,26.251,154.702
C06857=1071.734,136.529,-73.856,173.360,26.254,154.703
C06858=1071.740,136.778,-73.876,173.362,26.256,154.703
C06859=1071.745,137.027,-73.897,173.364,26.260,154.703
C06860=1071.751,137.276,-73.917,173.366,26.262,154.704
C06861=1071.757,137.526,-73.938,173.367,26.265,154.704
C06862=1071.763,137.774,-73.957,173.370,26.267,154.704
C06863=1071.768,138.023,-73.978,173.371,26.270,154.705
C06864=1071.773,138.273,-73.999,173.372,26.273,154.705
C06865=1071.780,138.522,-74.019,173.375,26.275,154.705
C06866=1071.786,138.771,-74.040,173.376,26.278,154.706
C06867=1071.792,139.019,-74.060,173.378,26.280,154.706
C06868=1071.797,139.269,-74.081,173.380,26.284,154.706
C06869=1071.803,139.518,-74.102,173.382,26.286,154.707
C06870=1071.809,139.767,-74.122,173.383,26.289,154.707
C06871=1071.814,140.016,-74.142,173.385,26.291,154.707
C06872=1071.819,140.265,-74.163,173.387,26.294,154.708
C06873=1071.826,140.514,-74.184,173.388,26.296,154.708
C06874=1071.831,140.763,-74.204,173.391,26.299,154.708
C06875=1071.837,141.013,-74.225,173.392,26.302,154.709
C06876=1071.842,141.262,-74.245,173.394,26.305,154.709
C06877=1071.849,141.511,-74.266,173.396,26.308,154.710
C06878=1071.854,141.760,-74.287,173.397,26.310,154.710
C06879=1071.859,142.009,-74.308,173.399,26.313,154.710
C06880=1071.865,142.258,-74.328,173.401,26.316,154.711
C06881=1071.871,142.507,-74.349,173.403,26.318,154.711
C06882=1071.877,142.789,-74.372,173.405,26.321,154.711
C06883=1071.884,143.072,-74.396,173.406,26.324,154.712
C06884=1071.890,143.354,-74.419,173.409,26.327,154.712
C06885=1071.897,143.637,-74.443,173.411,26.330,154.712
C06886=1071.902,143.886,-74.464,173.412,26.333,154.713
C06887=1071.908,144.134,-74.484,173.414,26.335,154.713
C06888=1071.914,144.383,-74.505,173.416,26.338,154.713
C06889=1071.919,144.633,-74.526,173.418,26.341,154.714
C06890=1071.925,144.882,-74.547,173.419,26.344,154.714
C06891=1071.930,145.131,-74.568,173.422,26.347,154.715
C06892=1071.937,145.380,-74.589,173.423,26.349,154.715
C06893=1071.942,145.629,-74.609,173.425,26.352,154.715
C06894=1071.948,145.879,-74.630,173.427,26.354,154.716
C06895=1071.954,146.127,-74.651,173.428,26.357,154.716
C06896=1071.959,146.376,-74.672,173.431,26.360,154.716
C06897=1071.966,146.625,-74.693,173.432,26.362,154.717
C06898=1071.971,146.874,-74.714,173.434,26.365,154.717
C06899=1071.977,147.123,-74.734,173.436,26.368,154.717
C06900=1071.983,147.373,-74.756,173.438,26.370,154.718
C06901=1071.988,147.622,-74.776,173.440,26.373,154.718
C06902=1071.994,147.870,-74.798,173.441,26.375,154.718
C06903=1071.999,148.120,-74.819,173.443,26.378,154.719
C06904=1072.006,148.368,-74.839,173.445,26.381,154.719
C06905=1072.012,148.618,-74.860,173.447,26.384,154.719
C06906=1072.017,148.867,-74.881,173.448,26.386,154.720
C06907=1072.022,149.116,-74.902,173.450,26.389,154.720
C06908=1072.029,149.365,-74.924,173.452,26.392,154.720
C06909=1072.034,149.614,-74.944,173.454,26.394,154.721
C06910=1072.040,149.863,-74.966,173.456,26.397,154.721
C06911=1072.045,150.112,-74.987,173.457,26.399,154.721
C06912=1072.051,150.361,-75.008,173.460,26.403,154.722
C06913=1072.057,150.610,-75.029,173.461,26.405,154.722
C06914=1072.062,150.859,-75.050,173.463,26.408,154.722
C06915=1072.068,151.108,-75.071,173.465,26.411,154.723
C06916=1072.074,151.357,-75.093,173.466,26.413,154.723
C06917=1072.079,151.606,-75.113,173.469,26.416,154.723
C06918=1072.085,151.855,-75.135,173.470,26.418,154.724
C06919=1072.091,152.104,-75.155,173.473,26.421,154.724
C06920=1072.097,152.354,-75.177,173.474,26.424,154.724
C06921=1072.102,152.602,-75.198,173.476,26.427,154.725
C06922=1072.107,152.852,-75.220,173.478,26.430,154.725
C06923=1072.113,153.101,-75.241,173.479,26.432,154.725
C06924=1072.119,153.349,-75.262,173.482,26.435,154.726
C06925=1072.125,153.598,-75.284,173.483,26.437,154.726
C06926=1072.130,153.848,-75.305,173.486,26.440,154.727
C06927=1072.136,154.097,-75.326,173.487,26.443,154.727
C06928=1072.142,154.345,-75.348,173.489,26.445,154.727
C06929=1072.148,154.595,-75.368,173.491,26.448,154.727
C06930=1072.153,154.844,-75.390,173.492,26.451,154.728
C06931=1072.159,155.093,-75.411,173.495,26.453,154.728
C06932=1072.165,155.341,-75.433,173.496,26.456,154.729
C06933=1072.171,155.591,-75.454,173.498,26.458,154.729
C06934=1072.176,155.840,-75.475,173.500,26.461,154.729
C06935=1072.182,156.089,-75.497,173.502,26.464,154.730
C06936=1072.187,156.338,-75.518,173.504,26.467,154.730
C06937=1072.193,156.587,-75.540,173.505,26.470,154.730
C06938=1072.199,156.835,-75.561,173.508,26.472,154.731
C06939=1072.203,157.085,-75.582,173.509,26.475,154.731
C06940=1072.210,157.334,-75.604,173.512,26.478,154.731
C06941=1072.215,157.583,-75.625,173.513,26.480,154.732
C06942=1072.221,157.832,-75.647,173.515,26.483,154.732
C06943=1072.228,158.081,-75.669,173.517,26.486,154.732
C06944=1072.232,158.330,-75.690,173.518,26.488,154.733
C06945=1072.239,158.579,-75.712,173.521,26.491,154.733
C06946=1072.244,158.861,-75.736,173.523,26.494,154.733
C06947=1072.251,159.143,-75.760,173.525,26.497,154.734
C06948=1072.258,159.425,-75.784,173.527,26.500,154.734
C06949=1072.264,159.707,-75.809,173.529,26.503,154.735
C06950=1072.270,159.957,-75.830,173.531,26.506,154.735
C06951=1072.275,160.205,-75.852,173.533,26.508,154.735
C06952=1072.281,160.455,-75.874,173.535,26.511,154.736
C06953=1072.287,160.703,-75.895,173.537,26.514,154.736
C06954=1072.293,160.952,-75.917,173.539,26.517,154.736
C06955=1072.298,161.202,-75.939,173.541,26.520,154.737
C06956=1072.304,161.450,-75.960,173.542,26.522,154.737
C06957=1072.309,161.700,-75.983,173.545,26.525,154.737
C06958=1072.315,161.948,-76.004,173.546,26.528,154.738
C06959=1072.320,162.198,-76.026,173.549,26.530,154.738
C06960=1072.326,162.446,-76.047,173.550,26.533,154.738
C06961=1072.331,162.696,-76.070,173.551,26.536,154.739
C06962=1072.337,162.944,-76.091,173.554,26.539,154.739
C06963=1072.343,163.193,-76.114,173.555,26.541,154.740
C06964=1072.348,163.442,-76.135,173.558,26.544,154.740
C06965=1072.354,163.691,-76.157,173.559,26.547,154.740
C06966=1072.358,163.940,-76.179,173.562,26.550,154.741
C06967=1072.365,164.189,-76.201,173.563,26.553,154.741
C06968=1072.369,164.438,-76.223,173.565,26.556,154.741
C06969=1072.376,164.687,-76.244,173.567,26.558,154.742
C06970=1072.380,164.936,-76.266,173.569,26.561,154.742
C06971=1072.387,165.185,-76.289,173.571,26.564,154.742
C06972=1072.392,165.434,-76.311,173.573,26.566,154.743
C06973=1072.397,165.683,-76.333,173.575,26.569,154.743
C06974=1072.403,165.932,-76.354,173.577,26.572,154.743
C06975=1072.408,166.181,-76.376,173.578,26.574,154.744
C06976=1072.415,166.430,-76.398,173.581,26.578,154.744
C06977=1072.419,166.679,-76.420,173.582,26.580,154.745
C06978=1072.425,166.928,-76.443,173.585,26.583,154.745
C06979=1072.431,167.177,-76.464,173.586,26.586,154.745
C06980=1072.436,167.425,-76.487,173.588,26.589,154.746
C06981=1072.442,167.675,-76.508,173.590,26.591,154.746
C06982=1072.448,167.924,-76.531,173.592,26.594,154.746
C06983=1072.453,168.172,-76.553,173.594,26.597,154.747
C06984=1072.459,168.422,-76.575,173.596,26.599,154.747
C06985=1072.464,168.670,-76.597,173.598,26.602,154.747
C06986=1072.470,168.920,-76.618,173.600,26.605,154.748
C06987=1072.476,169.169,-76.641,173.602,26.608,154.748
C06988=1072.481,169.417,-76.663,173.604,26.611,154.748
C06989=1072.487,169.667,-76.685,173.605,26.613,154.749
C06990=1072.492,169.915,-76.708,173.608,26.616,154.749
C06991=1072.497,170.164,-76.730,173.609,26.619,154.750
C06992=1072.504,170.413,-76.752,173.612,26.622,154.750
C06993=1072.509,170.662,-76.774,173.613,26.624,154.750
C06994=1072.515,170.912,-76.796,173.616,26.627,154.751
C06995=1072.520,171.160,-76.818,173.618,26.630,154.751
C06996=1072.526,171.409,-76.841,173.619,26.632,154.751
C06997=1072.532,171.658,-76.864,173.622,26.636,154.752
C06998=1072.537,171.907,-76.885,173.623,26.638,154.752
C06999=1072.543,172.156,-76.908,173.626,26.641,154.752
C07000=1072.548,172.405,-76.930,173.627,26.644,154.753
C07001=1072.554,172.654,-76.952,173.630,26.646,154.753
C07002=1072.560,172.902,-76.974,173.631,26.649,154.753
C07003=1072.565,173.152,-76.996,173.633,26.652,154.754
C07004=1072.571,173.401,-77.019,173.635,26.654,154.754
C07005=1072.577,173.650,-77.041,173.637,26.657,154.754
C07006=1072.582,173.898,-77.064,173.640,26.660,154.755
C07007=1072.589,174.147,-77.086,173.641,26.663,154.755
C07008=1072.594,174.396,-77.108,173.644,26.665,154.755
C07009=1072.600,174.645,-77.131,173.645,26.668,154.756
C07010=1072.606,174.927,-77.156,173.647,26.671,154.756
C07011=1072.613,175.209,-77.181,173.650,26.674,154.757
C07012=1072.619,175.491,-77.207,173.652,26.677,154.757
C07013=1072.626,175.773,-77.232,173.655,26.680,154.757
C07014=1072.630,176.021,-77.254,173.656,26.683,154.758
C07015=1072.637,176.270,-77.277,173.658,26.686,154.758
C07016=1072.643,176.519,-77.300,173.661,26.689,154.758
C07017=1072.648,176.768,-77.322,173.662,26.692,154.759
C07018=1072.654,177.017,-77.345,173.665,26.694,154.759
C07019=1072.660,177.266,-77.367,173.666,26.697,154.759
C07020=1072.665,177.515,-77.389,173.669,26.699,154.760
C07021=1072.671,177.764,-77.412,173.671,26.702,154.760
C07022=1072.677,178.013,-77.435,173.673,26.705,154.760
C07023=1072.683,178.262,-77.456,173.675,26.708,154.761
C07024=1072.688,178.511,-77.479,173.676,26.711,154.761
C07025=1072.694,178.760,-77.502,173.679,26.713,154.761
C07026=1072.700,179.008,-77.525,173.681,26.716,154.762
C07027=1072.706,179.258,-77.547,173.683,26.718,154.762
C07028=1072.711,179.506,-77.570,173.685,26.721,154.762
C07029=1072.717,179.755,-77.592,173.687,26.724,154.763
C07030=1072.723,180.004,-77.615,173.689,26.727,154.763
C07031=1072.729,180.253,-77.637,173.692,26.729,154.763
C07032=1072.735,180.502,-77.660,173.693,26.732,154.764
C07033=1072.740,180.751,-77.683,173.695,26.735,154.764
C07034=1072.746,181.000,-77.706,173.697,26.737,154.765
C07035=1072.752,181.248,-77.729,173.699,26.740,154.765
C07036=1072.758,181.498,-77.750,173.702,26.743,154.765
C07037=1072.764,181.747,-77.773,173.703,26.746,154.766
C07038=1072.769,181.995,-77.796,173.706,26.748,154.766
C07039=1072.775,182.244,-77.819,173.708,26.751,154.766
C07040=1072.781,182.493,-77.842,173.710,26.754,154.766
C07041=1072.787,182.742,-77.865,173.712,26.757,154.767
C07042=1072.793,182.991,-77.888,173.713,26.759,154.767
C07043=1072.799,183.240,-77.910,173.716,26.762,154.768
C07044=1072.804,183.489,-77.933,173.718,26.764,154.768
C07045=1072.810,183.738,-77.956,173.720,26.767,154.768
C07046=1072.816,183.987,-77.978,173.722,26.770,154.768
C07047=1072.822,184.235,-78.001,173.725,26.773,154.769
C07048=1072.828,184.484,-78.024,173.726,26.776,154.769
C07049=1072.834,184.733,-78.047,173.729,26.778,154.770
C07050=1072.839,184.982,-78.070,173.731,26.781,154.770
C07051=1072.845,185.231,-78.093,173.732,26.784,154.770
C07052=1072.849,185.480,-78.116,173.735,26.786,154.771
C07053=1072.855,185.728,-78.139,173.737,26.790,154.771
C07054=1072.861,185.977,-78.162,173.739,26.792,154.771
C07055=1072.867,186.226,-78.185,173.741,26.795,154.772
C07056=1072.872,186.475,-78.208,173.743,26.798,154.772
C07057=1072.877,186.724,-78.231,173.745,26.801,154.772
C07058=1072.883,186.973,-78.255,173.747,26.804,154.773
C07059=1072.889,187.222,-78.278,173.749,26.807,154.773
C07060=1072.894,187.471,-78.301,173.751,26.810,154.774
C07061=1072.900,187.720,-78.324,173.754,26.812,154.774
C07062=1072.906,187.969,-78.347,173.755,26.815,154.774
C07063=1072.911,188.217,-78.370,173.758,26.818,154.775
C07064=1072.916,188.467,-78.394,173.760,26.821,154.775
C07065=1072.922,188.716,-78.417,173.761,26.824,154.776
C07066=1072.928,188.964,-78.440,173.764,26.826,154.776
C07067=1072.934,189.213,-78.463,173.766,26.829,154.776
C07068=1072.939,189.462,-78.487,173.768,26.832,154.777
C07069=1072.944,189.711,-78.510,173.770,26.835,154.777
C07070=1072.950,189.960,-78.533,173.773,26.838,154.777
C07071=1072.955,190.208,-78.557,173.775,26.841,154.778
C07072=1072.961,190.457,-78.580,173.776,26.844,154.778
C07073=1072.967,190.706,-78.603,173.779,26.847,154.778
C07074=1072.973,190.987,-78.629,173.781,26.850,154.779
C07075=1072.979,191.268,-78.656,173.784,26.853,154.779
C07076=1072.986,191.550,-78.682,173.786,26.856,154.780
C07077=1072.992,191.832,-78.709,173.788,26.859,154.780
C07078=1072.998,192.080,-78.732,173.791,26.862,154.780
C07079=1073.004,192.329,-78.755,173.793,26.865,154.781
C07080=1073.009,192.578,-78.779,173.794,26.868,154.781
C07081=1073.014,192.827,-78.802,173.797,26.871,154.782
C07082=1073.020,193.075,-78.826,173.799,26.874,154.782
C07083=1073.025,193.325,-78.849,173.801,26.876,154.782
C07084=1073.031,193.573,-78.873,173.803,26.879,154.783
C07085=1073.037,193.822,-78.896,173.806,26.882,154.783
C07086=1073.042,194.071,-78.919,173.808,26.885,154.783
C07087=1073.048,194.319,-78.943,173.810,26.887,154.784
C07088=1073.054,194.568,-78.966,173.812,26.890,154.784
C07089=1073.060,194.817,-78.990,173.814,26.894,154.784
C07090=1073.066,195.066,-79.013,173.816,26.896,154.785
C07091=1073.071,195.315,-79.036,173.818,26.899,154.785
C07092=1073.077,195.564,-79.061,173.821,26.902,154.785
C07093=1073.082,195.813,-79.084,173.823,26.905,154.786
C07094=1073.088,196.061,-79.108,173.824,26.908,154.786
C07095=1073.093,196.310,-79.131,173.827,26.910,154.787
C07096=1073.100,196.559,-79.155,173.829,26.913,154.787
C07097=1073.105,196.808,-79.178,173.832,26.916,154.787
C07098=1073.111,197.057,-79.202,173.833,26.919,154.788
C07099=1073.116,197.306,-79.225,173.836,26.922,154.788
C07100=1073.122,197.554,-79.249,173.838,26.925,154.788
C07101=1073.128,197.802,-79.273,173.841,26.928,154.789
C07102=1073.134,198.052,-79.297,173.842,26.930,154.789
C07103=1073.140,198.301,-79.320,173.844,26.933,154.789
C07104=1073.145,198.550,-79.344,173.847,26.936,154.790
C07105=1073.151,198.798,-79.368,173.849,26.939,154.790
C07106=1073.156,199.047,-79.391,173.851,26.942,154.791
C07107=1073.162,199.296,-79.415,173.853,26.944,154.791
C07108=1073.168,199.545,-79.439,173.856,26.947,154.791
C07109=1073.173,199.794,-79.462,173.858,26.950,154.792
C07110=1073.179,200.042,-79.486,173.860,26.953,154.792
C07111=1073.185,200.291,-79.511,173.862,26.956,154.792
C07112=1073.191,200.540,-79.534,173.864,26.959,154.793
C07113=1073.197,200.789,-79.557,173.867,26.962,154.793
C07114=1073.202,201.037,-79.581,173.869,26.965,154.794
C07115=1073.209,201.287,-79.605,173.871,26.967,154.794
C07116=1073.214,201.535,-79.629,173.873,26.970,154.794
C07117=1073.220,201.784,-79.653,173.875,26.973,154.795
C07118=1073.226,202.033,-79.677,173.878,26.976,154.795
C07119=1073.232,202.282,-79.700,173.880,26.979,154.795
C07120=1073.237,202.530,-79.725,173.882,26.981,154.796
C07121=1073.243,202.779,-79.748,173.884,26.984,154.796
C07122=1073.249,203.028,-79.773,173.887,26.988,154.796
C07123=1073.254,203.276,-79.797,173.889,26.991,154.797
C07124=1073.259,203.526,-79.821,173.891,26.994,154.797
C07125=1073.265,203.774,-79.844,173.893,26.996,154.798
C07126=1073.271,204.023,-79.869,173.895,26.999,154.798
C07127=1073.276,204.272,-79.893,173.898,27.002,154.798
C07128=1073.282,204.520,-79.917,173.900,27.005,154.799
C07129=1073.288,204.769,-79.941,173.903,27.008,154.799
C07130=1073.294,205.018,-79.966,173.905,27.011,154.799
C07131=1073.299,205.267,-79.989,173.906,27.014,154.800
C07132=1073.305,205.515,-80.013,173.909,27.017,154.800
C07133=1073.311,205.765,-80.038,173.911,27.020,154.801
C07134=1073.316,206.013,-80.062,173.914,27.023,154.801
C07135=1073.321,206.262,-80.086,173.916,27.026,154.801
C07136=1073.328,206.511,-80.110,173.918,27.028,154.802
C07137=1073.333,206.760,-80.134,173.920,27.031,154.802
C07138=1073.357,207.800,-80.236,174.046,27.097,154.803
C07139=1073.367,208.216,-80.277,174.050,27.104,154.804
C07140=1073.377,208.633,-80.319,174.053,27.110,154.805
C07141=1073.386,209.048,-80.361,174.056,27.117,154.806
C07142=1073.396,209.466,-80.403,174.060,27.123,154.807
C07143=1073.402,209.714,-80.428,174.062,27.127,154.808
C07144=1073.407,209.963,-80.452,174.064,27.131,154.808
C07145=1073.413,210.212,-80.478,174.067,27.135,154.809
C07146=1073.419,210.461,-80.502,174.068,27.138,154.810
C07147=1073.425,210.709,-80.527,174.070,27.142,154.810
C07148=1073.431,210.958,-80.553,174.072,27.146,154.811
C07149=1073.437,211.207,-80.577,174.075,27.150,154.811
C07150=1073.442,211.455,-80.602,174.077,27.154,154.812
C07151=1073.448,211.704,-80.628,174.079,27.158,154.812
C07152=1073.454,211.953,-80.653,174.080,27.162,154.813
C07153=1073.459,212.201,-80.678,174.083,27.165,154.814
C07154=1073.466,212.450,-80.703,174.085,27.169,154.814
C07155=1073.472,212.699,-80.728,174.087,27.174,154.815
C07156=1073.477,212.947,-80.753,174.089,27.177,154.815
C07157=1073.483,213.196,-80.779,174.092,27.181,154.816
C07158=1073.489,213.445,-80.804,174.094,27.185,154.817
C07159=1073.494,213.693,-80.829,174.095,27.189,154.817
C07160=1073.500,213.942,-80.853,174.097,27.193,154.818
C07161=1073.506,214.191,-80.879,174.100,27.196,154.818
C07162=1073.511,214.439,-80.904,174.102,27.200,154.819
C07163=1073.518,214.688,-80.930,174.104,27.204,154.820
C07164=1073.523,214.937,-80.956,174.107,27.208,154.820
C07165=1073.529,215.186,-80.980,174.109,27.212,154.821
C07166=1073.535,215.434,-81.005,174.111,27.216,154.822
C07167=1073.540,215.683,-81.031,174.112,27.219,154.822
C07168=1073.546,215.932,-81.056,174.115,27.224,154.823
C07169=1073.552,216.180,-81.082,174.117,27.228,154.823
C07170=1073.557,216.428,-81.107,174.119,27.231,154.824
C07171=1073.564,216.677,-81.133,174.121,27.235,154.824
C07172=1073.570,216.926,-81.158,174.124,27.239,154.825
C07173=1073.575,217.175,-81.184,174.126,27.243,154.826
C07174=1073.581,217.423,-81.209,174.128,27.247,154.826
C07175=1073.587,217.671,-81.234,174.129,27.250,154.827
C07176=1073.592,217.920,-81.260,174.132,27.254,154.827
C07177=1073.599,218.169,-81.286,174.134,27.258,154.828
C07178=1073.604,218.417,-81.311,174.136,27.262,154.829
C07179=1073.610,218.666,-81.336,174.138,27.266,154.829
C07180=1073.616,218.915,-81.362,174.141,27.270,154.830
C07181=1073.621,219.164,-81.388,174.143,27.274,154.830
C07182=1073.628,219.412,-81.413,174.145,27.277,154.831
C07183=1073.634,219.661,-81.438,174.148,27.281,154.832
C07184=1073.639,219.909,-81.464,174.149,27.285,154.832
C07185=1073.645,220.158,-81.489,174.151,27.289,154.833
C07186=1073.650,220.407,-81.515,174.153,27.293,154.833
C07187=1073.657,220.656,-81.541,174.156,27.296,154.834
C07188=1073.663,220.904,-81.566,174.158,27.300,154.835
C07189=1073.668,221.153,-81.592,174.160,27.304,154.835
C07190=1073.675,221.401,-81.618,174.162,27.308,154.836
C07191=1073.684,221.822,-81.662,174.166,27.314,154.837
C07192=1073.694,222.243,-81.705,174.170,27.321,154.838
C07193=1073.704,222.664,-81.749,174.174,27.327,154.839
C07194=1073.713,223.085,-81.792,174.178,27.334,154.840
C07195=1073.719,223.333,-81.818,174.180,27.338,154.840
C07196=1073.725,223.582,-81.844,174.181,27.342,154.841
C07197=1073.730,223.831,-81.870,174.183,27.346,154.842
C07198=1073.737,224.079,-81.895,174.186,27.349,154.842
C07199=1073.742,224.328,-81.922,174.188,27.353,154.843
C07200=1073.748,224.576,-81.947,174.190,27.357,154.843
C07201=1073.753,224.825,-81.973,174.193,27.361,154.844
C07202=1073.759,225.073,-82.000,174.195,27.365,154.844
C07203=1073.765,225.322,-82.025,174.197,27.368,154.845
C07204=1073.771,225.571,-82.051,174.199,27.373,154.846
C07205=1073.777,225.819,-82.078,174.202,27.377,154.846
C07206=1073.783,226.068,-82.103,174.204,27.380,154.847
C07207=1073.788,226.317,-82.129,174.206,27.384,154.847
C07208=1073.794,226.565,-82.155,174.209,27.388,154.848
C07209=1073.800,226.814,-82.181,174.211,27.392,154.849
C07210=1073.806,227.062,-82.207,174.213,27.395,154.849
C07211=1073.812,227.311,-82.233,174.215,27.399,154.850
C07212=1073.818,227.559,-82.259,174.218,27.403,154.850
C07213=1073.824,227.808,-82.285,174.219,27.407,154.851
C07214=1073.829,228.057,-82.312,174.221,27.411,154.852
C07215=1073.836,228.305,-82.337,174.224,27.414,154.852
C07216=1073.841,228.554,-82.364,174.226,27.418,154.853
C07217=1073.847,228.803,-82.390,174.228,27.422,154.853
C07218=1073.853,229.051,-82.417,174.230,27.426,154.854
C07219=1073.859,229.300,-82.442,174.233,27.430,154.854
C07220=1073.865,229.548,-82.469,174.235,27.434,154.855
C07221=1073.870,229.797,-82.495,174.237,27.437,154.856
C07222=1073.876,230.045,-82.521,174.240,27.441,154.856
C07223=1073.882,230.294,-82.546,174.242,27.445,154.857
C07224=1073.888,230.542,-82.573,174.244,27.449,154.857
C07225=1073.894,230.791,-82.600,174.246,27.453,154.858
C07226=1073.899,231.040,-82.626,174.249,27.456,154.859
C07227=1073.905,231.288,-82.652,174.251,27.461,154.859
C07228=1073.911,231.536,-82.679,174.253,27.464,154.860
C07229=1073.916,231.785,-82.705,174.256,27.468,154.860
C07230=1073.922,232.034,-82.732,174.258,27.472,154.861
C07231=1073.929,232.282,-82.758,174.260,27.476,154.861
C07232=1073.934,232.531,-82.784,174.263,27.480,154.862
C07233=1073.940,232.780,-82.811,174.265,27.483,154.863
C07234=1073.946,233.028,-82.837,174.267,27.487,154.863
C07235=1073.952,233.277,-82.864,174.269,27.491,154.864
C07236=1073.957,233.526,-82.890,174.272,27.495,154.864
C07237=1073.963,233.774,-82.916,174.274,27.498,154.865
C07238=1073.969,234.022,-82.943,174.276,27.503,154.866
C07239=1073.974,234.271,-82.970,174.279,27.507,154.866
C07240=1073.980,234.519,-82.996,174.281,27.510,154.867
C07241=1073.986,234.767,-83.023,174.283,27.514,154.867
C07242=1073.991,235.016,-83.049,174.285,27.518,154.868
C07243=1074.001,235.429,-83.094,174.289,27.524,154.869
C07244=1074.011,235.842,-83.138,174.293,27.531,154.870
C07245=1074.020,236.254,-83.183,174.297,27.537,154.871
C07246=1074.030,236.667,-83.226,174.301,27.544,154.872
C07247=1074.036,236.915,-83.253,174.303,27.547,154.872
C07248=1074.042,237.164,-83.280,174.305,27.551,154.873
C07249=1074.048,237.412,-83.306,174.308,27.555,154.874
C07250=1074.053,237.660,-83.333,174.310,27.559,154.874
C07251=1074.059,237.910,-83.360,174.312,27.562,154.875
C07252=1074.065,238.158,-83.387,174.315,27.566,154.875
C07253=1074.070,238.406,-83.414,174.317,27.570,154.876
C07254=1074.076,238.655,-83.440,174.319,27.574,154.877
C07255=1074.082,238.903,-83.467,174.322,27.578,154.877
C07256=1074.088,239.152,-83.494,174.324,27.582,154.878
C07257=1074.094,239.401,-83.521,174.326,27.586,154.878
C07258=1074.100,239.648,-83.548,174.329,27.589,154.879
C07259=1074.106,239.897,-83.575,174.331,27.593,154.880
C07260=1074.112,240.146,-83.602,174.333,27.597,154.880
C07261=1074.117,240.394,-83.629,174.336,27.601,154.881
C07262=1074.123,240.643,-83.656,174.338,27.604,154.881
C07263=1074.129,240.891,-83.682,174.340,27.608,154.882
C07264=1074.135,241.140,-83.709,174.342,27.612,154.883
C07265=1074.141,241.389,-83.736,174.345,27.616,154.883
C07266=1074.146,241.637,-83.764,174.348,27.620,154.884
C07267=1074.152,241.885,-83.791,174.350,27.624,154.884
C07268=1074.159,242.134,-83.818,174.353,27.628,154.885
C07269=1074.164,242.382,-83.844,174.355,27.631,154.885
C07270=1074.170,242.630,-83.872,174.357,27.635,154.886
C07271=1074.176,242.880,-83.899,174.360,27.639,154.887
C07272=1074.182,243.128,-83.926,174.362,27.643,154.887
C07273=1074.188,243.376,-83.953,174.364,27.646,154.888
C07274=1074.193,243.624,-83.980,174.367,27.650,154.888
C07275=1074.199,243.873,-84.007,174.369,27.654,154.889
C07276=1074.204,244.122,-84.035,174.371,27.658,154.890
